(* CODESYS project MariaDB 1.0.1.6.library
   Description: connect to MariaDB read and write simple
      Impressed and helped with OSCAT
      www.oscat.de
   Version: 1.0.1.6
   Title: MariaDB
   Author: Stefan Dreyer
   DocFormat: reStructuredText
   Placeholder: MariaDB
   LanguageModelAttribute: qualified-access-only
   DefaultNamespace: MariaDB
   Company: Stefan Dreyer

Project tree, tasks and I/O mapping:
  libraries: CAA Types Extern, * (CAA Technical Workgroup); CAA Behaviour Model, * (CAA Technical Workgroup); CAA FB Factory, * (CAA Technical Workgroup); Time and Date, 3.5.7.0 (3S - Smart Software Solutions GmbH); SysFile, * (System); SysTypes Interfaces, * (System); Standard, * (System); SysMem, 3.5.12.0 (System); SysSocket, 3.5.15.0 (System); CmpErrors2 Interfaces, 3.5.15.0 (System); Raspberry I2C MUX, 1.0.1.2 (Stefan Dreyer); SysProcess, 3.5.16.0 (System); SysSem, 3.5.16.0 (System); Base Interfaces, 3.5.2.0 (System); BASIC, 3.3.4.0 (OSCAT); OSCAT Network Types, 1.0.0.2 (Stefan Dreyer); Common Helper for development, 1.1.0.6 (Stefan Dreyer); PRO JSON, 1.0.0.12 (Pro Electric)
  MariaDb/
    Structs/
      data type DATA_TO_DB
      data type VALUE_TO_DB_DATA_OFFLINE
      data type DB_SQL_DATA
      data type DATA_FROM_DB
      data type DB_IN_OUT
      data type SQL_ERROR
      data type PARAMETER_DB_DATA
      data type DATA_FOR_VALUE
      data type LOGGING_DATA
      data type COUNTER_TO_DB_DATA
    Function Blocks/
      function block HANDLE_SQL_DB [ST]: SQL_RESPONSE_COMMON
      function block VALUE_TO_DB [ST]: PUSH_LOCAL_BUFFER, SET_DB_REQUEST_FOR_PW_CONFIG, CHECK_DATA_FROM_DB, DO_SQL_DATA, SET_CONFIG_VALUE
      function block TIME_DATE_IMPULS [ST]
      function block MARIADB_CONTROL [ST]
      function block SQL_BASE [ST]: PUT_SQL_TO_BUFFER, CREATE_SQL, SAVE_SQL_ERROR, GET_INDEX_DATA_FIELDS_SQL_RESPONSE, CHECK_EOF_PAKET, DO_SQL_DATA, SET_DB_IN_OUT_PTR
      function block LOGGING_TO_DB [ST]: DO_SQL_DATA, PUSH_LOCAL_BUFFER, SetConfig
      function block PARAMETER_DB [ST]: CHECK_DIFF_VAR, DO_SQL_DATA, GET_PAGE_ADRESS_EEPROM, CHECK_DATA_FROM_DB, CHECK_DATA_FROM_EEPROM
      function block STRING_DB [ST]: CHECK_DIFF_VAR, DO_SQL_DATA, GET_PAGE_ADRESS_EEPROM, CHECK_DATA_FROM_DB, CHECK_DATA_FROM_EEPROM
      function block COUNTER_DB [ST]: SET_CONFIG_COUNTER, PUSH_LOCAL_BUFFER, DO_SQL_DATA
      function block VALUE_TO_DB_AUTO_ID [ST]: PUSH_LOCAL_BUFFER, SET_DB_REQUEST_FOR_PW_CONFIG, CHECK_DATA_FROM_DB, DO_SQL_DATA, SET_CONFIG_VALUE, SET_CONFIG_VALUE_LEVELS, SetRealFaktor
      function block LOGGING_TO_DB_AUTO_ID [ST]: DO_SQL_DATA, PUSH_LOCAL_BUFFER, CHECK_DATA_FROM_DB, SET_DB_REQUEST_FOR_TEXT_CONFIG
      function block VALUE_TO_DB_AUTO_ID_ANY [ST]: PUSH_LOCAL_BUFFER, SET_DB_REQUEST_FOR_PW_CONFIG, CHECK_DATA_FROM_DB, DO_SQL_DATA, SET_CONFIG_VALUE, SET_CONFIG_VALUE_LEVELS
      function block VALUE_TO_DB_AUTO_ID_JSON [ST]: FB_Init
      function block COUNTER_DB_AUTO_ID [ST]: SET_CONFIG_COUNTER, PUSH_LOCAL_BUFFER, DO_SQL_DATA, CHECK_DATA_FROM_DB, SET_DB_REQUEST_FOR_COUNTER_NUM
    GlobalConstants/
      global variables MyConstants
    Types/
      data type SQL_COMMANDS
      data type MYSQL_COM
      data type DB_RESPONSE
    Functions/
      function GET_STRING_DATE [ST]
      function GET_STRING_FROM_RESPONSE [ST]
*)

// MariaDb/Structs/DATA_TO_DB
TYPE DATA_TO_DB :

STRUCT
	//ID of SQL FB to store or of request form DB
	FB_ID:UINT;
	//SQL number
	SQL_NO: INT;//Number of SQL
	//SQL for DB
	SQL_STRING:STRING(MyConstants.COM_STRING_SIZE);
END_STRUCT
END_TYPE

// MariaDb/Structs/VALUE_TO_DB_DATA_OFFLINE
TYPE VALUE_TO_DB_DATA_OFFLINE :
STRUCT
	VALUE:CommonTypesAndFunctions.ALL_TYPES_UNION;
	VALUE_TIME:DT;
END_STRUCT
END_TYPE

// MariaDb/Types/SQL_COMMANDS
{attribute 'qualified_only'}
{attribute 'strict'}
TYPE SQL_COMMANDS :
(
	SEND_PW := 0, SEND_REQUEST_GET_PW_CONFIG := 1, WRITE_LOGGING_TEXT := 2, GET_PARAMETER_VALUE := 3, SET_PARAMETER_VALUE := 4,
	GET_PARAMETER_STRING := 5, SET_PARAMETER_STRING := 6, PUT_COUNTER_TO_DB := 7, PUT_COUNTER_TO_DB_WITH_FACTOR := 8,
	SEND_REQUEST_GET_PW_CONFIG_INSTANCE_NAME := 9, GET_LOGGING_TEXT := 10, CREATE_NEW_SENSOR_ENTRY := 11,
	CREATE_NEW_TEXT_ENTRY := 12, SEND_PW_PROZEDUR := 13, SEND_COUNTER_PROZEDUR := 14, GET_COUNTER_NUM := 15,
	CREATE_NEW_COUNTER_ENTRY := 16
);
END_TYPE

// MariaDb/Structs/DB_SQL_DATA
TYPE DB_SQL_DATA :
STRUCT
//All Infos for an SQL Insert/request for very small SQL!
SQL_TEMPLATE:STRING(255);
SQL_KEYWORDS:ARRAY[0..MyConstants.SQL_MAX_KEYWORDS] OF STRING;
SQL_RESPONSE_FIELDS:INT;//Zero means no Answer expected

END_STRUCT
END_TYPE

// MariaDb/Types/MYSQL_COM
TYPE MYSQL_COM :
STRUCT
	S_BUF : OSCAT_NETWORK_TYPES.NETWORK_BUFFER;
	R_BUF : OSCAT_NETWORK_TYPES.NETWORK_BUFFER;
	SQL_CON : BOOL;
	SQL_URL : STRING(OSCAT_BASIC.STRING_LENGTH);
	SQL_PACKET_NO : BYTE;
	TIMEOUT : TIME;
	DNS_IP4 : DWORD;
	SQL_RCV_STATE : BYTE;
	ERROR_C : DWORD;
	ERROR_T : BYTE;
	RESPONSE : POINTER TO STRING;//pointer for String for Response
	RESPONSE_SIZEOF:UINT;//Max Size of String
	
(* revision history
ks	27. oct. 2012	rev 1.0
	original version
*)
(*
Update from Stefan Dreyer for prozessing responses
01.05.2017
*)
END_STRUCT
END_TYPE

// MariaDb/Structs/DATA_FROM_DB
TYPE DATA_FROM_DB :
STRUCT
	FB_ID:UINT;//ID of SQL Data
	//SQL number
	SQL_NO: INT;
	RESPONSE_TYPE:INT;//Type of response
	DATA_FROM_DB:ARRAY[0..OSCAT_NETWORK_TYPES.NETWORK_BUFFER_LONG_SIZE]OF BYTE;
	SQL_ERROR:SQL_ERROR;
END_STRUCT
END_TYPE

// MariaDb/Structs/DB_IN_OUT
TYPE DB_IN_OUT :
STRUCT
	IN:DATA_TO_DB;
	OUT:DATA_FROM_DB;
	IMP:BOOL;//1s impulse
	SYSTEM_TIME:DT;//Time on SYSTEM
	TIME_IO:BOOL;//TIME IS I.O.
	SQL_CONNECTED:BOOL;
	FB_NO_AUTO:UINT;//
	TD_TIME:OSCAT_BASIC.SDT;
	pendingData:UDINT;
END_STRUCT
END_TYPE

// MariaDb/Types/DB_RESPONSE
{attribute 'qualified_only'}
{attribute 'strict'}
TYPE DB_RESPONSE :
(
	ERROR := -1, OK := 1, DATA_RETURNED := 2
);
END_TYPE

// MariaDb/Structs/SQL_ERROR
TYPE SQL_ERROR :
STRUCT
	SQL_ERROR:STRING(255);//SQL ERROR FROM DB
	SQL_NO:INT;
	SQL_ERROR_TIME:DT;
END_STRUCT
END_TYPE

// MariaDb/Structs/PARAMETER_DB_DATA
TYPE PARAMETER_DB_DATA:
STRUCT
	DATA_EEPROM:CommonTypesAndFunctions.EEPROM_DATA;
	STRING_COUNT:UINT := 200;
	HAS_DB: BOOL;
	HAS_EEPROM: BOOL;
	DB_HAS_PRIORITY: BOOL;
	EEPROM_HAS_PRIORITY: BOOL;

END_STRUCT
END_TYPE

// MariaDb/Structs/DATA_FOR_VALUE
TYPE DATA_FOR_VALUE :
STRUCT
	//name aof Value
	Name:STRING[30];
	//Value itself
	Value: CommonTypesAndFunctions.ALL_TYPES_UNION;
	//type of this value
	TypeOfValue:IBaseLibrary.TypeClass;
	//Number of Value in DB
	ValueNum:UINT;
	//Impulse for value
	ImpValue:BOOL;
END_STRUCT
END_TYPE

// MariaDb/Structs/LOGGING_DATA
TYPE LOGGING_DATA :
STRUCT
	//Time of event
	TimeToLog:DT;
	//positiv or negativ edge
	POrN:BOOL;
	
END_STRUCT
END_TYPE

// MariaDb/Structs/COUNTER_TO_DB_DATA
TYPE COUNTER_TO_DB_DATA :
STRUCT
	VALUE_TIME:DT;
END_STRUCT
END_TYPE

// MariaDb/GlobalConstants/MyConstants
{attribute 'qualified_only'}
VAR_GLOBAL CONSTANT
	FB_BUFFER_SIZE:UINT:=20000;
	COM_STRING_SIZE:UINT:=255;
	SQL_MAX_KEYWORDS:UINT:=10;
	SQL_KEYWORDS_SIZE:UINT:=20;
	SQL_DATA_BUFFER_SIZE:UINT:=200;
	NETWORK_BUFFER_LONG_SIZE:UINT:=4095;
	SQL_RESPONSE_MAX_STRING_SIZE:UINT:=200;
	SQL_LENGTH_FIELD_PAKET:UINT:=5;
	SQL_SIZE_OF_HEADER:UINT:=4;
	SQL_SIZE_OF_EOF_PAKET:UINT:=9;
	SQL_OFFSET_DATA_PAKET:UINT:=4;
SQLS: ARRAY[0..16] OF DB_SQL_DATA:=[
					(*0*)
					(SQL_TEMPLATE:='insert into home.allsensors values("valueWhen", SENSOR, VALUE)',
					SQL_KEYWORDS := ['valueWhen','SENSOR','VALUE'], SQL_RESPONSE_FIELDS := 0),
					(*1*)
					(SQL_TEMPLATE:='select intervall, factor, deltaVar from home.sensors where sensorNum = SENSOR',
					SQL_KEYWORDS := ['SENSOR'], SQL_RESPONSE_FIELDS := 3),
					(*2*)
					(SQL_TEMPLATE:='insert into home.logging(textWhen, text, id_text) values("WHEN1", "TEXT", "ID_TEX_T")',
					SQL_KEYWORDS := ['WHEN1', 'TEXT','ID_TEX_T'], SQL_RESPONSE_FIELDS := 0),
					(*3*)
					(SQL_TEMPLATE:='select value from home.param_value where INDEX = INDEX_NO',
					SQL_KEYWORDS := ['INDEX_NO'], SQL_RESPONSE_FIELDS := 1),
					(*4*)
					(SQL_TEMPLATE:='replace into home.param_value values(INDEX, VALUE)',
					SQL_KEYWORDS := ['INDEX', 'VALUE'], SQL_RESPONSE_FIELDS := 0),
					(*5*)
					(SQL_TEMPLATE:='select string from home.param_string where INDEX = INDEX_NO',
					SQL_KEYWORDS := ['INDEX_NO'], SQL_RESPONSE_FIELDS := 1),
					(*6*)
					(SQL_TEMPLATE:='replace into home.param_string values(INDEX, "STRING")',
					SQL_KEYWORDS := ['INDEX', 'STRING'], SQL_RESPONSE_FIELDS := 0),
					(*7*)
					(SQL_TEMPLATE:='insert into home.allsensors values("valueWhen", SENSOR, 1)',
					SQL_KEYWORDS := ['valueWhen','SENSOR'], SQL_RESPONSE_FIELDS := 0),
					(*8*)
					(SQL_TEMPLATE:='INSERT INTO home.allsensors(valueWhen, sensor, value) VALUES("valueWhen1", NUM, FACTOR / TIMESTAMPDIFF(SECOND,(SELECT * FROM (SELECT MAX(valueWhen) from home.allsensors WHERE sensor = NUM)t),"valueWhen1"))',
					SQL_KEYWORDS := ['valueWhen1','NUM','FACTOR'], SQL_RESPONSE_FIELDS := 0),
					(*9*)
					(SQL_TEMPLATE:='select intervall, factor, deltaVar, sensorNum from home.sensors where Instance = "FBName"',
					SQL_KEYWORDS := ['FBName'], SQL_RESPONSE_FIELDS := 4),
					(*10*)
					(SQL_TEMPLATE:='select texte.text, texte.index from home.texte where Instance = "FBName"',
					SQL_KEYWORDS := ['FBName'], SQL_RESPONSE_FIELDS := 2),
					(*11*)
					(SQL_TEMPLATE:='INSERT INTO home.sensors(description,sensorNum,INSTANCE,Factor) VALUES("NBEZ",(SELECT*FROM home.nextn),"NINSTANCE","NFAKTOR")',
					SQL_KEYWORDS := ['NBEZ', 'NINSTANCE', 'NFAKTOR'], SQL_RESPONSE_FIELDS := 0),
					(*12*)
					(SQL_TEMPLATE:='INSERT INTO home.texte(TEXT, INSTANCE) VALUES("NTEXT", "NINSTANCE")',
					SQL_KEYWORDS := ['NTEXT', 'NINSTANCE'], SQL_RESPONSE_FIELDS := 0),
					(*13*)
					(SQL_TEMPLATE:='CALL home.InsertValue("valueWhen", SENSOR, VALUE)',
					SQL_KEYWORDS := ['valueWhen', 'SENSOR', 'VALUE'], SQL_RESPONSE_FIELDS := 0),
					(*14*)
					(SQL_TEMPLATE:='CALL home.InsertCounter("valueWhen", SENSOR, FAKTOR)',
					SQL_KEYWORDS := ['valueWhen', 'SENSOR', 'FAKTOR'], SQL_RESPONSE_FIELDS := 1),
					(*15*)
					(SQL_TEMPLATE:='select sensorNum from home.sensors where Instance = "FBName"',
					SQL_KEYWORDS := ['FBName'], SQL_RESPONSE_FIELDS := 1),
					(*16*)
					(SQL_TEMPLATE:='INSERT INTO home.sensors(description,sensorNum,INSTANCE,factor) VALUES("NBEZ",(SELECT*FROM home.nextnc),"NINSTANCE","NFAKTOR")',
					SQL_KEYWORDS := ['NBEZ', 'NINSTANCE', 'NFAKTOR'], SQL_RESPONSE_FIELDS := 0)];
END_VAR

// MariaDb/Function Blocks/HANDLE_SQL_DB
FUNCTION_BLOCK HANDLE_SQL_DB  
VAR_IN_OUT
	SQL_INFO : OSCAT_NETWORK_TYPES.MYSQL_INFO;
	DB_IN_OUT:DB_IN_OUT;
END_VAR
VAR_INPUT
	ENABLE : BOOL;
	URL : STRING(OSCAT_BASIC.STRING_LENGTH);
	TIMEOUT : TIME;
END_VAR
VAR_OUTPUT
	ERROR_C : DWORD;
	ERROR_T : BYTE;
END_VAR
VAR
	DT_Maria:TIME_DATE_IMPULS;
	MARIADB_CONTROL: MARIADB_CONTROL;
	step : INT;
	snd_size : INT;
	sql_command : BYTE;
	next_step : INT;
	i1 : INT;
	i2 : INT;
	size_of_string_in_response:UINT;
	len_paket:UDINT;
	id1:UDINT;
	com: MYSQL_COM;
	
	//ID of FB from request
	FB_ID_REQUEST : UINT;
	//Number of actuel SQL
	AKT_SQL_NO : INT;
	
		
	T_SPS_LAST_REQUEST_STARTET:DWORD;
	TIME_LAST_REQUEST:DWORD;
	TIME_LAST_REQUEST_MIN:DWORD:=16#FFFFFFFF;
	TIME_LAST_REQUEST_MAX:DWORD;
	SQLS_PER_SECOND:DWORD;
	TIME_TO_NEW_REQUEST:DWORD;
	SQLS_DONE_IO:DWORD;
	T_SPS_LAST_REQUEST_FINISHED:DWORD;
	CYCLE_TIME:DWORD;
	LAST_CYCLE_TIME:DWORD;
	pendingData:UDINT;
	
END_VAR


DB_IN_OUT.FB_NO_AUTO := 0;//reset FB number
pendingData:= DB_IN_OUT.pendingData;
DB_IN_OUT.pendingData:= 0; 
CYCLE_TIME := OSCAT_BASIC.T_PLC_MS() - LAST_CYCLE_TIME;
LAST_CYCLE_TIME := OSCAT_BASIC.T_PLC_MS();
//get system time and so one
DT_Maria(
	DB_IN_OUT:= DB_IN_OUT);
DB_IN_OUT.IMP := DT_Maria.IMP;
DB_IN_OUT.SYSTEM_TIME := DT_Maria.DT_OUT;
DB_IN_OUT.TIME_IO := DT_Maria.TIME_VAILID;

CASE step OF

00:	IF ENABLE THEN
		COM.SQL_URL := URL;
		COM.TIMEOUT := TIMEOUT;
		step := 10;
		COM.SQL_CON := TRUE;
		
	END_IF;
10:	IF SQL_INFO.SQL_CONNECTED THEN
		step := 40;
	END_IF;
40:	


	IF DB_IN_OUT.IN.FB_ID > 0 AND step = 40 THEN (* Neue Datenreihe(n) vorhanden *)
		(*insert Dato only in step 40!*)

		//start sql command
		sql_command := BYTE#3;
		//store sql in DB Buffer
		OSCAT_BASIC._STRING_TO_BUFFER(str:=DB_IN_OUT.IN.SQL_STRING,pos:=5,pt:=ADR(COM.S_BUF.BUFFER),size:=SIZEOF(COM.S_BUF.BUFFER)); (* String in puffer kopieren *)
		FB_ID_REQUEST := DB_IN_OUT.IN.FB_ID;
		AKT_SQL_NO := DB_IN_OUT.IN.SQL_NO;
		next_step := 40;
		snd_size := 5 + OSCAT_BASIC.LEN(STR:= DB_IN_OUT.IN.SQL_STRING) ;
		T_SPS_LAST_REQUEST_STARTET := OSCAT_BASIC.T_PLC_MS();
		TIME_TO_NEW_REQUEST := OSCAT_BASIC.T_PLC_MS() - T_SPS_LAST_REQUEST_FINISHED;
	END_IF

	IF NOT  ENABLE THEN 	(* LOG-Trigger verarbeiten *)
		COM.SQL_CON := FALSE; (* MySQL Verbindung beenden *)
		step := 0;
	END_IF;

(* ~~~~~~~~~~~~~~~~~~~~~~ *)

199:IF COM.SQL_RCV_STATE = BYTE#1 THEN (* OK *)
		IF MyConstants.SQLS[AKT_SQL_NO].SQL_RESPONSE_FIELDS > 0 THEN//last sql command was request
			//Parse response
			IF COM.R_BUF.BUFFER[4] = MyConstants.SQLS[AKT_SQL_NO].SQL_RESPONSE_FIELDS THEN
				//response have the right number of fields
				//put recive buffer to out bufferNETWORK_BUFFER_LONG_SIZE
				DB_IN_OUT.OUT.DATA_FROM_DB := COM.R_BUF.BUFFER;
				DB_IN_OUT.OUT.SQL_NO:= AKT_SQL_NO;
				DB_IN_OUT.OUT.FB_ID := FB_ID_REQUEST;
				DB_IN_OUT.OUT.RESPONSE_TYPE := DB_RESPONSE.DATA_RETURNED;
			ELSE	
				//wrong response!
				step := 0;//ERROR
			END_IF

		END_IF
		step := next_step;
		SQLS_DONE_IO := SQLS_DONE_IO + 1;
		SQL_RESPONSE_COMMON(DB_IN_OUT:=DB_IN_OUT);
	ELSIF COM.SQL_RCV_STATE = BYTE#2 THEN  (* FEHLER *)
		//step := 0;
		DB_IN_OUT.OUT.SQL_ERROR.SQL_ERROR := SQL_INFO.SQL_ERROR;
		DB_IN_OUT.OUT.SQL_ERROR.SQL_NO := AKT_SQL_NO;
		DB_IN_OUT.OUT.SQL_ERROR.SQL_ERROR_TIME := DB_IN_OUT.SYSTEM_TIME;
		DB_IN_OUT.OUT.FB_ID := FB_ID_REQUEST;
		DB_IN_OUT.OUT.RESPONSE_TYPE := DB_RESPONSE.ERROR;
		COM.SQL_RCV_STATE := BYTE#1;//recive zurücksetzten
		SQL_RESPONSE_COMMON(DB_IN_OUT:=DB_IN_OUT);
	END_IF;

END_CASE;

(* ########################## *)
(* SQL-Kommando ausführen *)
IF sql_command > BYTE#0 THEN

	COM.S_BUF.SIZE := INT_TO_UINT(snd_size);
	snd_size := 0;
	
	i2 := UINT_TO_INT(COM.S_BUF.SIZE) - 1; (* alle " zeichen mit ' ersetzen *)
	FOR i1 := 5 TO i2 DO
		IF COM.S_BUF.BUFFER[i1] = BYTE#34 THEN
			COM.S_BUF.BUFFER[i1] := BYTE#39;
		END_IF;
	END_FOR;

	COM.S_BUF.BUFFER[4] := sql_command;
	COM.SQL_PACKET_NO := BYTE#255;
	sql_command := BYTE#0;
	step := 199;
END_IF;

(* ########################## *)

MARIADB_CONTROL(COM:= COM, INFO:=SQL_INFO);
ERROR_C := COM.ERROR_C;
ERROR_T := COM.ERROR_T;

IF COM.ERROR_T > BYTE#0 THEN  (* FEHLER *)
	step := 0;
END_IF;
//put status to SQLs
DB_IN_OUT.SQL_CONNECTED := SQL_INFO.SQL_CONNECTED;
(* ########################## *)

(* revision history
ks	20. apr. 2012	rev 1.0
	original version

*)

METHOD SQL_RESPONSE_COMMON : BOOL
VAR_IN_OUT
	DB_IN_OUT:DB_IN_OUT;
END_VAR
VAR_INPUT
END_VAR
//Eingänge zurück setzten
DB_IN_OUT.IN.FB_ID := 0;
DB_IN_OUT.IN.SQL_NO := 0;
TIME_LAST_REQUEST := OSCAT_BASIC.T_PLC_MS() - T_SPS_LAST_REQUEST_STARTET;
T_SPS_LAST_REQUEST_FINISHED := OSCAT_BASIC.T_PLC_MS();
TIME_LAST_REQUEST_MIN := MIN(TIME_LAST_REQUEST, TIME_LAST_REQUEST_MIN);
TIME_LAST_REQUEST_MAX := MAX(TIME_LAST_REQUEST, TIME_LAST_REQUEST_MAX);
SQLS_PER_SECOND := REAL_TO_DWORD(1/(DWORD_TO_REAL(TIME_LAST_REQUEST)/1000));
END_METHOD

END_FUNCTION_BLOCK

// MariaDb/Function Blocks/MARIADB_CONTROL
FUNCTION_BLOCK MARIADB_CONTROL
(*
update for MariaDB an not only insert and update(select with !1! result), by Stefan Dreyer
update für MariaDB um nicht nur insert und update sondern auch select(mit max einer antwort!) zu ermöglichen von Stefan Dreyer
*)
VAR_IN_OUT
	COM : MYSQL_COM;
	INFO : OSCAT_NETWORK_TYPES.MYSQL_INFO;
END_VAR
VAR_OUTPUT
END_VAR
VAR
	IP_C : CommonTypesAndFunctions.IP_C_EXT;
	URL_DATA : OSCAT_NETWORK_TYPES.url;
	IPC : CommonTypesAndFunctions.IP_CONTROL;

	step : INT;
	snd_step : INT;
	TON_WAIT : OSCAT_BASIC.TON;
	last_step : INT;
	idx1 : INT;
	idx2 : INT;
	idx3 : INT;
	dw_tmp : DWORD;
	timeout1 : TIME;
	timeout2 : TIME;
	ip_c_red_disable : BOOL;
	auth_password : STRING(64);
	auth_run : BOOL;
	MYSQL_AUTH : OSCAT_NETWORK_TYPES.MYSQL_AUTH;
	scramble1_buffer : ARRAY [0..19] OF BYTE;
	scramble2_buffer : ARRAY [0..19] OF BYTE;
	charset_number : BYTE := 16#08;
	max_packet_size : DWORD := 1024;
	client_flags : DWORD := 16#0003_8601;
	sResultIP : STRING; // IP-Address behind hostname
	(*
	LOG_MSG : LOG_MSG;
	_debug_enable : BOOL := TRUE;
	*)

	nop: INT;
END_VAR

(*
version 1.0		16. apr. 2012
programmer		ks
tested by		ks

MYSQL_CONTROL führt einen SQL Befehl auf einem MySQL-Server durch 
*)

IF com.ERROR_C <> 0 THEN
 step := step;
END_IF 

CASE step OF

00:	IF COM.SQL_CON THEN
		timeout1 := MAX(T#10s,COM.TIMEOUT);
		timeout2 := timeout1 + T#1s;
		INFO.SQL_ERROR := '';
		COM.ERROR_C := DWORD#0;
		COM.ERROR_T := BYTE#0;
		URL_DATA := OSCAT_NETWORK_TYPES.STRING_TO_URL(STR:=COM.SQL_URL,DEFAULT_PROTOCOL:='',DEFAULT_PATH:='/');
		step := 10;
	END_IF;

10:	IF CommonTypesAndFunctions.ResolveIPAddr(sHost:= URL_DATA.DOMAIN, sIPResult:= ADR(sResultIP)) = CmpErrors.Errors.ERR_OK THEN
		step := 20;
	ELSE
		step := 980;
	END_IF

20:	(* MariaDB Steuerkanal einrichten *)
	IF URL_DATA.PORT = WORD#0 THEN
		URL_DATA.PORT := WORD#3306; (* Standard Port *)
	END_IF;
	IP_C.C_PORT := URL_DATA.PORT; (* Portnummer eintragen *)
  	IP_C.C_IP := OSCAT_NETWORK_TYPES.IP4_DECODE(sResultIP); (* IP eintragen *)
  	IP_C.C_MODE := BYTE#0; (* Mode: TCP+ACTIV+PORT *)
  	IP_C.TIME_RESET := TRUE; (* Zeitueberwachung rücksetzen *)
  	IP_C.C_ENABLE := TRUE; (* Verbindungsaufbau freigeben *)
  	IP_C.R_OBSERVE := TRUE; (* Empfangsueberwachung *)
	COM.R_BUF.SIZE := UINT#0;
	COM.SQL_RCV_STATE := BYTE#0;
	step := 30;

30:	IF COM.SQL_RCV_STATE = BYTE#1 THEN
		INFO.SERVER_PROTOCOL_VERSION := COM.R_BUF.BUFFER[4];

		(* ende markierung von string server_version suchen *)
		idx2 := UINT_TO_INT(COM.R_BUF.SIZE) - 1;
		FOR idx1 := 5 TO idx2 DO
			IF COM.R_BUF.BUFFER[idx1] = BYTE#0 THEN EXIT; END_IF;
		END_FOR;
		idx1 := idx1 + 5; (* terminierung und thread-id überspringen *)

		FOR idx2:=0 TO 7 DO	(* Byte 0-7 *)
			scramble1_buffer[idx2] := COM.R_BUF.BUFFER[idx1];
			idx1 := idx1 + 1;
		END_FOR;
		idx1 := idx1 + 1;
		idx2 := idx1 + 1;
		INFO.SERVER_CAPABILITIES := OSCAT_BASIC.WORD_OF_BYTE(COM.R_BUF.BUFFER[idx2], COM.R_BUF.BUFFER[idx1]);
		idx1 := idx1 + 2;
		INFO.SERVER_LANGUAGE := COM.R_BUF.BUFFER[idx1];
		idx1 := idx1 + 1;
		idx2 := idx1 + 1;
		INFO.SERVER_STATUS := OSCAT_BASIC.WORD_OF_BYTE(COM.R_BUF.BUFFER[idx2], COM.R_BUF.BUFFER[idx1]);
		idx1 := idx1 + 15;

		FOR idx2:=8 TO 19 DO	(* Byte 8-19 *)
			scramble1_buffer[idx2] := COM.R_BUF.BUFFER[idx1];
			idx1 := idx1 + 1;
		END_FOR;

		IF INFO.SERVER_PROTOCOL_VERSION < BYTE#10 THEN  (* Error: protocol version zu niedrig *)
			COM.ERROR_T := BYTE#2;
			COM.ERROR_C := DWORD#1;
			step := 980;
		ELSIF URL_DATA.PASSWORD = '' THEN
			step := 50;
		ELSE
			auth_password := URL_DATA.PASSWORD;
			auth_run := TRUE;
			step := 40;
		END_IF;
	END_IF;

40:	MYSQL_AUTH(RUN:= auth_run,PASSWORD:= auth_password ,MESSAGE:= scramble1_buffer,SCRAMBLE:= scramble2_buffer);
	IF NOT auth_run THEN
		step := 50;
	END_IF;

50: (* Client Authentication Packet *)
	(* Byte 0-3 werden später eingetragen *)
	COM.S_BUF.BUFFER[04] := OSCAT_BASIC.BYTE_OF_DWORD(client_flags, BYTE#0); (* client_flags *)
	COM.S_BUF.BUFFER[05] := OSCAT_BASIC.BYTE_OF_DWORD(client_flags, BYTE#1);
	COM.S_BUF.BUFFER[06] := OSCAT_BASIC.BYTE_OF_DWORD(client_flags, BYTE#2);
	COM.S_BUF.BUFFER[07] := OSCAT_BASIC.BYTE_OF_DWORD(client_flags, BYTE#3);
	COM.S_BUF.BUFFER[08] := OSCAT_BASIC.BYTE_OF_DWORD(max_packet_size, BYTE#0); (* max_packet_size *)
	COM.S_BUF.BUFFER[09] := OSCAT_BASIC.BYTE_OF_DWORD(max_packet_size, BYTE#1);
	COM.S_BUF.BUFFER[10] := OSCAT_BASIC.BYTE_OF_DWORD(max_packet_size, BYTE#2);
	COM.S_BUF.BUFFER[11] := OSCAT_BASIC.BYTE_OF_DWORD(max_packet_size, BYTE#3);
	COM.S_BUF.BUFFER[12] := charset_number; (* charset_number *)
	FOR idx1 := 13 TO 35 DO (* 23 bytes filler always 0x00.. *)
		COM.S_BUF.BUFFER[idx1] := BYTE#0;
	END_FOR;
	idx3 := OSCAT_BASIC.LEN(URL_DATA.USER);
	FOR idx2 :=1 TO idx3 DO
		COM.S_BUF.BUFFER[idx1] := OSCAT_BASIC.CODE(URL_DATA.USER, idx2);
		idx1 := idx1 + 1;
	END_FOR;
	COM.S_BUF.BUFFER[idx1] := BYTE#0; (* String terminierung eintragen *)
	idx1 := idx1 + 1;
	IF OSCAT_BASIC.LEN(URL_DATA.PASSWORD) = 0 THEN
		COM.S_BUF.BUFFER[idx1] := BYTE#0; (* scramble_buff length *)
	ELSE
		COM.S_BUF.BUFFER[idx1] := BYTE#20; (* scramble_buff length *)
		FOR idx2 :=0 TO 19 DO
			idx1 := idx1 + 1;
			COM.S_BUF.BUFFER[idx1] := scramble2_buffer[idx2];
		END_FOR;
	END_IF;
	COM.S_BUF.SIZE  := INT_TO_UINT(idx1 + 1); (* Sendelänge eintragen *)

	step := 60;

60:	IF COM.SQL_RCV_STATE = BYTE#1 THEN
		INFO.SQL_CONNECTED := TRUE;
		step := 300;
	END_IF;

(* ================================================== *)

300:	step := UINT_TO_INT(SEL(COM.SQL_CON,700,310)); (* Schritt-Selektion *)

310:	step := 300; (* dummy step *)

(* ================================================== *)

700: (* COM_QUIT *)
	COM.S_BUF.BUFFER[04] := BYTE#1; (* 0x01 COM_QUIT mysql_close *)
	COM.S_BUF.SIZE := UINT#5; (* Sendelänge eintragen *)
	COM.SQL_PACKET_NO := BYTE#255;
	ip_c_red_disable := TRUE;
	step := 710;

710:	IF IP_C.C_STATE = BYTE#0 THEN (* Verbindung durch SQL-Server beendet ? *)
		step := 980;
	END_IF;

(* ================================================== *)

980:IP_C.C_ENABLE := FALSE; (* MYSQL Steuerkanal schliessen *)
	ip_c_red_disable := FALSE;
	INFO.SQL_CONNECTED := FALSE;
	//COM.SQL_CON := FALSE;
	COM.S_BUF.SIZE := UINT#0;
	COM.R_BUF.SIZE := UINT#0;
	snd_step := 0;
	step := 990;
	(*####################  DEBUG-MESSAGE  ###################################*)
	(*IF _debug_enable THEN
		LOG_CL.NEW_MSG := 'QUIT: ERROR CODE >~1< TYPE >~2<';
		LOG_CL.PRINTF[1] := DWORD_TO_STRH(COM.ERROR_C);
		LOG_CL.PRINTF[2] := BYTE_TO_STRING(COM.ERROR_T);
		LOG_MSG();
	END_IF;*)
	(*########################################################################*)

990:IF IP_C.C_STATE = BYTE#0 THEN
		step := 0;
	END_IF;

END_CASE;

(* ++++++++++++++++++++++++++++++++++++++++++++++++++++++++++ *)

IF step >= 30 THEN
	IF COM.R_BUF.SIZE >= UINT#3 AND COM.SQL_RCV_STATE = BYTE#0 THEN (* Daten wurden empfangen ? *)
		(*hier Prüfung für OK und ERROR Paket, immer nur ein Paket*)
		(*Zu erledigen, Error an SQL Ersteller zurück liefern und SQL Verbindung nicht trennen*)
		IF DWORD_TO_UINT(OSCAT_BASIC.DWORD_OF_BYTE(BYTE#0, COM.R_BUF.BUFFER[2], COM.R_BUF.BUFFER[1], COM.R_BUF.BUFFER[0])) + UINT#4 = COM.R_BUF.SIZE THEN
			COM.SQL_PACKET_NO := COM.R_BUF.BUFFER[3];
			IF COM.R_BUF.BUFFER[4] = BYTE#16#FF THEN
				idx2 := 13; (* Error String - Erstes Zeichen *)
				idx3 := UINT_TO_INT(COM.R_BUF.SIZE) - 1; (* Error String - Letztes Zeichen *)
				FOR idx1 := idx2 TO idx3 DO (* alle ' durch ´ ersetzen *)
					IF COM.R_BUF.BUFFER[idx1] = BYTE#39 THEN
						COM.R_BUF.BUFFER[idx1] := BYTE#96;
					END_IF;
				END_FOR;
				INFO.SQL_ERROR := OSCAT_BASIC.BUFFER_TO_STRING(PT:=ADR(COM.R_BUF.BUFFER),SIZE:=COM.R_BUF.SIZE,START:=INT_TO_UINT(idx2),STOP:=INT_TO_UINT(idx3));
				COM.SQL_RCV_STATE := BYTE#2;
				COM.R_BUF.SIZE := UINT#0; (* Empfangsbuffer nach Fehler rücksetzen *)
				
			ELSE
				(*hier OK Paket*)
				COM.SQL_RCV_STATE := BYTE#1;
				(*####################  DEBUG-MESSAGE  ###################################*)
				(*IF _debug_enable THEN
					LOG_CL.NEW_MSG := 'RCV: size >~1<';
					LOG_CL.PRINTF[1] := UINT_TO_STRING(COM.R_BUF.SIZE);
					LOG_MSG();
				END_IF;*)
				(*########################################################################*)
			END_IF;
		ELSE
		//hier mehr Paket Antworten bearbeite.	
		//Parsen der Antworten je nach request

		//Hier oder im Aufruf????  
		//Abarbeitung im Aufruf

		END_IF;
		IF DWORD_TO_UINT(OSCAT_BASIC.DWORD_OF_BYTE(BYTE#0, COM.R_BUF.BUFFER[2], COM.R_BUF.BUFFER[1], COM.R_BUF.BUFFER[0])) = 1 THEN//recived response with data
			COM.SQL_RCV_STATE := BYTE#1;
			
		
		END_IF;
		IP_C.R_OBSERVE := FALSE;
	END_IF;
END_IF;

(* automatisches Datensenden *)

CASE snd_step OF

00:	IF step >= 20 AND COM.S_BUF.SIZE > UINT#0 THEN
		dw_tmp := UINT_TO_DWORD(COM.S_BUF.SIZE - UINT#4); (* packet_length *)
		COM.S_BUF.BUFFER[0] := OSCAT_BASIC.BYTE_OF_DWORD(dw_tmp, BYTE#0);
		COM.S_BUF.BUFFER[1] := OSCAT_BASIC.BYTE_OF_DWORD(dw_tmp, BYTE#1);
		COM.S_BUF.BUFFER[2] := 0;
		COM.SQL_PACKET_NO := COM.SQL_PACKET_NO + 1;
		COM.S_BUF.BUFFER[3] := COM.SQL_PACKET_NO;

		IP_C.R_OBSERVE := TRUE;
		COM.R_BUF.SIZE := UINT#0; (* Empfangsbuffer rücksetzen *)
		COM.SQL_RCV_STATE := BYTE#0;

	        (*####################  DEBUG-MESSAGE  ###################################*)
	        (*IF _debug_enable THEN
	          LOG_CL.NEW_MSG := 'SND: size >~1<';
	          LOG_CL.PRINTF[1] := UINT_TO_STRING(COM.S_BUF.SIZE);
	          LOG_MSG();
	        END_IF;*)
	        (*########################################################################*)

		snd_step := 10;
	END_IF;

10:	IF COM.S_BUF.SIZE = UINT#0 THEN (* warten bis alle daten gesendet sind *)
		snd_step := 0;
	END_IF;

END_CASE;

(* Globale Fehlerbehandlung für Haupt-Routine *)
IF COM.ERROR_T = BYTE#0 AND step > 20 THEN (* noch kein Fehler gespeichert und Hauptroutine aktiv *)
	IF IP_C.ERROR > DWORD#0 AND IP_C.C_ENABLE AND NOT IP_C.TIME_RESET THEN  (* IP Control *)
		IF ip_c_red_disable = FALSE OR IP_C.ERROR <> DWORD#16#FD000000 THEN
			COM.ERROR_C := IP_C.ERROR;
			COM.ERROR_T := BYTE#2;
			step := 980;
		END_IF;
	END_IF;
END_IF;

IF TON_WAIT.Q THEN (* Ablaufstörung - Schrittkette *)
	COM.ERROR_C := INT_TO_DWORD(step); (* aktuellen Schritt eintragen *)
	COM.ERROR_T := BYTE#5;
	step := 980;
END_IF;

(* ######################################################## *)

IPC(IP:= DWORD#0, PORT:= WORD#0 , TIME_OUT:= timeout1, IP_C:= IP_C, S_BUF:= COM.S_BUF, R_BUF:= COM.R_BUF); (* MYSQL Steuerkanal *)

TON_WAIT(IN:=step = last_step AND step > 0,PT:=timeout2);
last_step := step;


(* revision history
ks	20. apr. 2012	rev 1.0
	original version

*)

END_FUNCTION_BLOCK

// MariaDb/Function Blocks/TIME_DATE_IMPULS
FUNCTION_BLOCK TIME_DATE_IMPULS
VAR_IN_OUT
	DB_IN_OUT:DB_IN_OUT;
END_VAR
VAR_INPUT
END_VAR
VAR_OUTPUT
	DT_OUT:DT; //Date an Time
	IMP: BOOL; //1s impulse
	TIME_VAILID: BOOL := FALSE; //Time is Valid
	TD:OSCAT_BASIC.SDT;
END_VAR
VAR
	RT_SYS:RTCLK.GetDateAndTime;
	RT:OSCAT_BASIC.RTC_2;
	DT_OLD:DT;
	GET_TIME: BOOL := TRUE;
	TIME_READED: BOOL;
	TIMEZONE:RTCLK.PERIODE;
	ReReadTime: BOOL;
	ReReadErrorTime:TON;
	ReReadTimeCycle:TON;
END_VAR

RT_SYS(xExecute := GET_TIME);
IF RT_SYS.xDone THEN
	GET_TIME := FALSE;
	IF	RT_SYS.dtDateAndTime < DT#1980-01-01-00:00:00 THEN
		//Keine Valide Uhr auf Raspi!
		ReReadTime := TRUE;
		TIME_VAILID := FALSE;
	ELSE
		TIME_READED := TRUE;
		TIMEZONE := RT_SYS.eTimezone;
		ReReadTime := FALSE;
		TIME_VAILID := TRUE;
	END_IF
END_IF
//Zykliches neulsesen der Uhrzeit
ReReadTimeCycle(in := (TIME_VAILID AND NOT GET_TIME), PT:= T#30M);
IF ReReadTimeCycle.Q THEN
	GET_TIME := TRUE;//try again to read Time	
END_IF


//Neulesezeit nach Error bearbeiten:
ReReadErrorTime(in:=ReReadTime, pt:=T#1S);
IF ReReadErrorTime.Q THEN
	ReReadTime := FALSE;
	GET_TIME := TRUE;//try again to read Time
END_IF
//Realtime Clock bearbeiten // Setzten
RT(set := TIME_READED, SDT := RT_SYS.dtDateAndTime, OFS := 60, DEN:=TRUE);
TIME_READED := FALSE;
//Date and time from oscat fb
DT_OUT:=RT.LOCAL_DT;
//check for second impuls
IF DT_OLD <> DT_OUT THEN
	DT_OLD := DT_OUT;
	imp := TRUE;
ELSE
	imp := FALSE;
END_IF
//make Time for OSCAT functions
TD := OSCAT_BASIC.DT_TO_SDT(DTI:= DT_OUT);

DB_IN_OUT.IMP := IMP;
DB_IN_OUT.SYSTEM_TIME := DT_OUT;
DB_IN_OUT.TD_TIME := TD;
DB_IN_OUT.TIME_IO := TIME_VAILID;

END_FUNCTION_BLOCK

// MariaDb/Function Blocks/VALUE_TO_DB
(*HOWTO
this function controls the sending of process data to DB.
if the queue to db is full it stors the value and date local.
if this local buffer is full, the request is dropt.
the id of the call aof this function must be greater then 0 for detection if the queue to db is empty

*)


FUNCTION_BLOCK VALUE_TO_DB EXTENDS SQL_BASE
VAR_INPUT
	
END_VAR
VAR_OUTPUT
END_VAR
VAR_IN_OUT
	
END_VAR
VAR
	//pointer to extern value
	PointerToValue:CommonTypesAndFunctions.ALL_TYPES_UNION_POINTER;
	
	//Value itself
	Value:CommonTypesAndFunctions.ALL_TYPES_UNION;
	//Impulse for value
	ImpValue:BOOL;
	//Value Name
	Name:STRING(50);
	//type of this value
	TypeOfValue:IBaseLibrary.TypeClass;
	//Number of Value in DB
	ValueNum:UINT;
	//stored Data from request
	DATA_REQUEST:DATA_TO_DB;
	//buffer for DB Offline
	BUFFER:ARRAY[0..MyConstants.FB_BUFFER_SIZE] OF VALUE_TO_DB_DATA_OFFLINE;
	

	//Delta time
	DELTA_T:UINT := 60;
	//Time var for DELTA_T
	DELTA_T_VAR:UINT;
	//type of var to save
	VAR_TYPE:UINT;
	//delta value
	DeltaVar:UINT:=1;
	//Last value of VAR send to DB
	LAST_VALUE:CommonTypesAndFunctions.ALL_TYPES_UNION;
	//request by time and Value given
	REQUEST_INSERT: BOOL;
	//Faktor for real for fix komma
	RealFaktor:UINT:=1;
	//check config from DB every....s
	CHECK_DB_CONFIG:UINT:=300;
	//var for waiting to check
	CHECK_DB_CONFIG_VAR:UINT;
	
	FL_IMP_TO_DB:R_TRIG;
	// set to true, if config is reaced
	configDone: BOOL;

END_VAR

//set right config status to parent
SQLInvalid := NOT configDone;
SQL_NO:=SQL_COMMANDS.SEND_PW_PROZEDUR;//set SQL no for super^()
SUPER^();
//if not config, then leave, do this after super so we calc correct FB numbers
IF ValueNum = 0 OR NOT DbPointerIo THEN RETURN; END_IF;


//just work when Time is i.o.
IF NOT DB_IN_OUT^.TIME_IO THEN RETURN; END_IF
//get value from pointer
Value := CommonTypesAndFunctions.GetValueFromPointer(PointerToValue:= PointerToValue, TypeOfValue:= TypeOfValue);
//Check if a config request is todo
IF DATA_REQUEST.FB_ID <> 0 AND DB_IN_OUT^.IN.FB_ID = 0 THEN
	DB_IN_OUT^.IN := DATA_REQUEST;
	
	DATA_REQUEST.FB_ID := 0;//delete request
END_IF

CHECK_DATA_FROM_DB();

//no second imp, nothing to do...
IF NOT DB_IN_OUT^.IMP  THEN
	RETURN;
END_IF
SET_DB_REQUEST_FOR_PW_CONFIG();
//check time over or impulse
FL_IMP_TO_DB(CLK:= ImpValue);
IF DELTA_T_VAR >0 THEN
	DELTA_T_VAR := DELTA_T_VAR -1;
	IF NOT FL_IMP_TO_DB.Q THEN
		RETURN;
	END_IF
END_IF
//check delta V
REQUEST_INSERT := CommonTypesAndFunctions.CheckDeltaValue(Value:= Value, DeltaVar:= DeltaVar, Faktor:= RealFaktor, LastValue:= LAST_VALUE, TypeOfValue:= TypeOfValue);
//nothing todo...
IF NOT REQUEST_INSERT THEN RETURN; END_IF
//we have an request, so first set new intervall
DELTA_T_VAR := DELTA_T - 1;

//push every Data to local buffer, may we lose an cycle but we have only on place to db 
//check buffer to DB free
	//push to lokal buffer
	//if buffer is full drop request
IF BUFFER_INDEX < MyConstants.FB_BUFFER_SIZE THEN
	PUSH_LOCAL_BUFFER();
END_IF

REQUEST_INSERT := FALSE;

METHOD PRIVATE PUSH_LOCAL_BUFFER
VAR_INPUT
END_VAR
VAR_IN_OUT
END_VAR
IF BUFFER_INDEX < MyConstants.FB_BUFFER_SIZE - 1 THEN 
	BUFFER[BUFFER_INDEX].value := Value;
	BUFFER[BUFFER_INDEX].value_time := DB_IN_OUT^.SYSTEM_TIME;
	BUFFER_INDEX := BUFFER_INDEX + 1; 
END_IF
IF BUFFER_INDEX > MaxBuffer THEN
	MaxBuffer := BUFFER_INDEX;
END_IF
END_METHOD

METHOD PRIVATE SET_DB_REQUEST_FOR_PW_CONFIG
VAR_IN_OUT
END_VAR
//check if time is over
IF CHECK_DB_CONFIG_VAR > 0 THEN
	CHECK_DB_CONFIG_VAR := CHECK_DB_CONFIG_VAR - 1;
	RETURN;	
END_IF
IF NOT DB_IN_OUT^.SQL_CONNECTED THEN RETURN; END_IF
//set new intervall
CHECK_DB_CONFIG_VAR := CHECK_DB_CONFIG;

//now put the request to DB

SQL_VALUES[0] := UINT_TO_STRING(ValueNum);

DATA_REQUEST := PUT_SQL_TO_BUFFER(SQL_NO:=SQL_COMMANDS.SEND_REQUEST_GET_PW_CONFIG);
END_METHOD

METHOD PRIVATE CHECK_DATA_FROM_DB
VAR_IN_OUT
END_VAR
VAR
	i:UINT;
END_VAR
IF DB_IN_OUT^.OUT.FB_ID = DB_IN_OUT^.FB_NO_AUTO THEN
	//got my request back	
	i := GET_INDEX_DATA_FIELDS_SQL_RESPONSE(src:=ADR(DB_IN_OUT^.OUT.DATA_FROM_DB),SQL_COMMANDS.SEND_REQUEST_GET_PW_CONFIG);
	IF i = 0 THEN 
	
		SQL_ERROR.SQL_ERROR := 'no data to Sensor';

		//SQL I.O. but no data 
	ELSE
		//parse first data
		DELTA_T := LIMIT(1, STRING_TO_WORD(GET_STRING_FROM_RESPONSE(SRC:=ADR(DB_IN_OUT^.OUT.DATA_FROM_DB), SIZE:=SIZEOF(DB_IN_OUT^.OUT.DATA_FROM_DB),I:=i)), 65000);
		//Set var to new value to prevent high times in some cases
		DELTA_T_VAR := LIMIT(1, DELTA_T, DELTA_T_VAR);
		//get faktor for Real values
		RealFaktor := LIMIT(1, STRING_TO_WORD(GET_STRING_FROM_RESPONSE(SRC:=ADR(DB_IN_OUT^.OUT.DATA_FROM_DB), SIZE:=SIZEOF(DB_IN_OUT^.OUT.DATA_FROM_DB),I:=i)),100);
		//get min delta for values
		DeltaVar := LIMIT(1, STRING_TO_WORD(GET_STRING_FROM_RESPONSE(SRC:=ADR(DB_IN_OUT^.OUT.DATA_FROM_DB), SIZE:=SIZEOF(DB_IN_OUT^.OUT.DATA_FROM_DB),I:=i)),1000);
	END_IF
	DB_IN_OUT^.OUT.FB_ID := 0;//delete response
	configDone := TRUE;
END_IF
END_METHOD

METHOD PRIVATE DO_SQL_DATA
VAR_INPUT
END_VAR
SQL_VALUES[0] := GET_STRING_DATE(BUFFER[BUFFER_INDEX].value_time);
SQL_VALUES[1] := UINT_TO_STRING(ValueNum);
SQL_VALUES[2] := CommonTypesAndFunctions.GetValueStringFaktor(VALUE:= BUFFER[BUFFER_INDEX].value, TypeOfValue:= TypeOfValue, RealFaktor:= TO_INT(RealFaktor), DecimalPlace:= 0);
END_METHOD

METHOD SET_CONFIG_VALUE
VAR_INPUT
	//Name of Value
	Name:STRING[50];
	//type of this value
	TypeOfValue:IBaseLibrary.TypeClass;
	//Number of Value in DB
	ValueNum:UINT;
	//pointer to value
	PointerToValue:CommonTypesAndFunctions.ALL_TYPES_UNION_POINTER;
	//Pointer to DB Data
	DB_IN_OUT:POINTER TO DB_IN_OUT;
	
END_VAR
THIS^.Name := Name;
	
THIS^.TypeOfValue:=TypeOfValue;
	
THIS^.ValueNum := ValueNum;

THIS^.PointerToValue := PointerToValue;

THIS^.SET_DB_IN_OUT_PTR(DB_IN_OUT);
END_METHOD

END_FUNCTION_BLOCK

// MariaDb/Function Blocks/SQL_BASE
FUNCTION_BLOCK SQL_BASE
VAR_IN_OUT
	
END_VAR
VAR_OUTPUT
END_VAR
VAR
	//referenz to DB Struct
	DB_IN_OUT:POINTER TO DB_IN_OUT;
	//SQL VALUES for SQL string
	SQL_VALUES:ARRAY[0..MyConstants.SQL_MAX_KEYWORDS-1] OF STRING;
	SQL_ERROR:SQL_ERROR;
	
	//index for use of buffer, point to first empty element
	BUFFER_INDEX:UINT;
	//Number of SQL to do From Child, to do the correct SQL replacment 
	SQL_NO:INT;
	//set to true, if something is missing for SQL replacment, so, you can wait till its done
	SQLInvalid: BOOL:=FALSE;
	//Set to true if get DB Pointer 
	DbPointerIo:BOOL;
	//max use of locak buffer
	MaxBuffer:UINT;
	//Instance name
	MyName:CommonTypesAndFunctions.GetInstanceName;
	//get config name String
	getConfigName:STRING;
	
END_VAR

IF not DbPointerIo THEN RETURN; END_IF
	

DB_IN_OUT^.FB_NO_AUTO := DB_IN_OUT^.FB_NO_AUTO + 1;
//add pending Data
DB_IN_OUT^.pendingData:= DB_IN_OUT^.pendingData + BUFFER_INDEX;
SAVE_SQL_ERROR();//check if i did get an SQL ERROR
IF SQLInvalid THEN RETURN; END_IF
//POP from buffer for all childs
IF BUFFER_INDEX > 0 AND DB_IN_OUT^.IN.FB_ID = 0 THEN
	//here pop buffer
	BUFFER_INDEX := BUFFER_INDEX - 1;
	//call child
	DO_SQL_DATA();
	//call child
	DB_IN_OUT^.IN:=PUT_SQL_TO_BUFFER(SQL_NO:=SQL_NO);
END_IF

METHOD PUT_SQL_TO_BUFFER : DATA_TO_DB
VAR_IN_OUT
END_VAR
VAR_INPUT
	SQL_NO:INT;
END_VAR
PUT_SQL_TO_BUFFER.FB_ID := DB_IN_OUT^.FB_NO_AUTO;
PUT_SQL_TO_BUFFER.SQL_NO := SQL_NO;
PUT_SQL_TO_BUFFER.SQL_STRING := CREATE_SQL(SQL_NO:=SQL_NO);
END_METHOD

METHOD CREATE_SQL : String(255)
VAR_INPUT
	SQL_NO:INT;
END_VAR
VAR
	i:INT;
END_VAR
i := 0;
CREATE_SQL := MyConstants.SQLS[SQL_NO].SQL_TEMPLATE;

WHILE MyConstants.SQLS[SQL_NO].SQL_KEYWORDS[i] <> '' DO
	CREATE_SQL := OSCAT_BASIC.REPLACE_ALL(str:=CREATE_SQL, src:=MyConstants.SQLS[SQL_NO].SQL_KEYWORDS[i], rep:=SQL_VALUES[i]);
	i := i + 1;
END_WHILE
END_METHOD

METHOD SAVE_SQL_ERROR : String(255)
VAR_INPUT
END_VAR
VAR_IN_OUT
END_VAR
IF DB_IN_OUT^.FB_NO_AUTO = DB_IN_OUT^.OUT.FB_ID AND DB_IN_OUT^.OUT.RESPONSE_TYPE = DB_RESPONSE.ERROR THEN
	SQL_ERROR := DB_IN_OUT^.OUT.SQL_ERROR;
	DB_IN_OUT^.OUT.FB_ID := 0;//delete response
END_IF
END_METHOD

METHOD GET_INDEX_DATA_FIELDS_SQL_RESPONSE : uint;//found index, if 0 sql i.o. but no data

VAR_INPUT
	src : POINTER TO ARRAY[0..32767]OF BYTE; 
	ID_REQUEST: INT;
END_VAR

VAR
	id1: UINT;
	i1: INT;
	len_paket: UINT;
END_VAR
//now get index of Values paket
GET_INDEX_DATA_FIELDS_SQL_RESPONSE := 0; //if zero, nothing found
//first search first EOF Paket
id1 := MyConstants.SQL_LENGTH_FIELD_PAKET;//second paket index after number of fields
FOR i1 := 0 TO MyConstants.SQLS[ID_REQUEST].SQL_RESPONSE_FIELDS - 1 DO
	len_paket := DWORD_TO_UINT(OSCAT_BASIC.DWORD_OF_BYTE(BYTE#0, src^[+id1+2], src^[id1+1], src^[id1]));
	id1 := id1 + len_paket + MyConstants.SQL_SIZE_OF_HEADER(*SIZE OF HEADER*);
END_FOR
//now i got through all colum definition pakets
//now im must see an eof paket
//paket size should be 5 and EOF MARKER should be 16#fe
IF CHECK_EOF_PAKET(src:=src, i:=id1) THEN
	id1 := id1 + MyConstants.SQL_SIZE_OF_EOF_PAKET;//Index to next paket, Data Paket
END_IF
//if the next paket is an eof paket, no data have been received
IF NOT CHECK_EOF_PAKET(src:=src, i:=id1) THEN
	GET_INDEX_DATA_FIELDS_SQL_RESPONSE := id1 + MyConstants.SQL_OFFSET_DATA_PAKET;				
END_IF
END_METHOD

METHOD CHECK_EOF_PAKET : bool
VAR_INPUT
	src:POINTER TO ARRAY[0..32000]OF BYTE;
	i:UINT;
END_VAR
CHECK_EOF_PAKET :=src^[i] = BYTE#5  AND src^[i+4] =16#FE;
END_METHOD

METHOD DO_SQL_DATA
VAR_INPUT
END_VAR
//just leave Empty, Overwrite in your implementation
END_METHOD

METHOD SET_DB_IN_OUT_PTR : INT
VAR_INPUT
	DB_IN_OUT:POINTER TO DB_IN_OUT;
END_VAR
THIS^.DB_IN_OUT := DB_IN_OUT;
DbPointerIo := TRUE;
END_METHOD

END_FUNCTION_BLOCK

// MariaDb/Functions/GET_STRING_FROM_RESPONSE
FUNCTION GET_STRING_FROM_RESPONSE : STRING(MyConstants.SQL_RESPONSE_MAX_STRING_SIZE)
VAR_INPUT
	SRC:POINTER TO ARRAY[0..32767]OF BYTE;
	SIZE: UINT;
END_VAR
VAR_IN_OUT
	I:UINT;
END_VAR
VAR
END_VAR

GET_STRING_FROM_RESPONSE := OSCAT_BASIC.BUFFER_TO_STRING(PT:=SRC, SIZE:=SIZE,START:=i+1,STOP:=i+1+(SRC^[i] - 1));
i := i + 1 + SRC^[i];

END_FUNCTION

// MariaDb/Functions/GET_STRING_DATE
FUNCTION GET_STRING_DATE : string
VAR_INPUT
DATE_IN:DT;
END_VAR
VAR
END_VAR

GET_STRING_DATE := DT_TO_STRING(DATE_IN);
GET_STRING_DATE := OSCAT_BASIC.RIGHT(STR := GET_STRING_DATE, SIZE := 19);
GET_STRING_DATE := OSCAT_BASIC.REPLACE(STR1:= GET_STRING_DATE, STR2:= ' ', L:= 1, P:= 11);

END_FUNCTION

// MariaDb/Function Blocks/LOGGING_TO_DB
FUNCTION_BLOCK LOGGING_TO_DB EXTENDS SQL_BASE
VAR_INPUT
	//TRIGGER: BOOL;
	Trigger:BOOL;
END_VAR
VAR_OUTPUT
END_VAR
VAR
	BUFFER:ARRAY[0..MyConstants.FB_BUFFER_SIZE] OF LOGGING_DATA;
	
	P_TRIGGER:Standard.R_TRIG;
	N_TRIGGER:Standard.F_TRIG;
	TextOn :STRING(200);
	TextOff :STRING(200);
	IdTextOn:UINT;
	IdTextOff:UINT;
	

END_VAR

SQL_NO:=SQL_COMMANDS.WRITE_LOGGING_TEXT;//set SQL no for super^()

SUPER^();
//my work isnt vailid without time... or DB Pointer
IF NOT DbPointerIo THEN RETURN; END_IF
IF NOT DB_IN_OUT^.TIME_IO THEN RETURN; END_IF

P_TRIGGER(CLK:= Trigger);
N_TRIGGER(CLK:= Trigger);

IF BUFFER_INDEX < MyConstants.FB_BUFFER_SIZE AND ((P_TRIGGER.Q AND IdTextOn > 0)OR (N_TRIGGER.Q AND IdTextOff > 0)) THEN
	PUSH_LOCAL_BUFFER();
END_IF

METHOD DO_SQL_DATA
VAR_INPUT
END_VAR
SQL_VALUES[0] := GET_STRING_DATE(BUFFER[BUFFER_INDEX].TimeToLog);
IF BUFFER[BUFFER_INDEX].POrN THEN //check if event was positiv or negativ
	SQL_VALUES[1] := TextOn;
	SQL_VALUES[2] := UINT_TO_STRING(IdTextOn);
ELSE
	SQL_VALUES[1] := TextOff;	
	SQL_VALUES[2] := UINT_TO_STRING(IdTextOff);
END_IF
END_METHOD

METHOD PUSH_LOCAL_BUFFER
VAR_INPUT
END_VAR
VAR_IN_OUT
	//DB_IN_OUT:DB_IN_OUT;
END_VAR
IF BUFFER_INDEX < MyConstants.FB_BUFFER_SIZE - 1 THEN
	BUFFER[BUFFER_INDEX].TimeToLog := DB_IN_OUT^.SYSTEM_TIME;
	BUFFER[BUFFER_INDEX].POrN := Trigger;
END_IF

BUFFER_INDEX := BUFFER_INDEX + 1; 

IF BUFFER_INDEX > MaxBuffer THEN
	MaxBuffer := BUFFER_INDEX;
END_IF
END_METHOD

METHOD SetConfig
VAR_INPUT
	TextOn:STRING(200);
	TextOff:STRING(200);

	IdTextOn:UINT;
	IdTextOff:UINT;
END_VAR
THIS^.TextOn := TextOn;
THIS^.TextOff := TextOff;
THIS^.IdTextOn := IdTextOn;
THIS^.IdTextOff := IdTextOff;
END_METHOD

END_FUNCTION_BLOCK

// MariaDb/Function Blocks/PARAMETER_DB
//this FB saves an Parameter to DB and/or to EEPROM

FUNCTION_BLOCK PARAMETER_DB EXTENDS SQL_BASE
VAR_IN_OUT
	PARAM:CommonTypesAndFunctions.ALL_TYPES_UNION;
	PARAM_DATA:PARAMETER_DB_DATA;
END_VAR
VAR_INPUT

	PARAMETER_NO:UINT;

END_VAR
VAR_OUTPUT
	VAR_VAILID:BOOL; //Datwas read by DB or EEPROM
END_VAR
VAR
	LAST_VALUE:CommonTypesAndFunctions.ALL_TYPES_UNION;
	SQL_COMMAND:INT;
	INIT_DONE:BOOL;
	BUFFER:ARRAY[0..0] OF CommonTypesAndFunctions.ALL_TYPES_UNION;
	SAVE_PARAM: BOOL;
	EEPROM_SAVE_DONE: BOOL;
	DB_SAVE_DONE: BOOL;
	LOCAL_PARAM:CommonTypesAndFunctions.ALL_TYPES_UNION;
	
	LOAD_AT_BOOT_DONE: BOOL := FALSE;
	
	VALUE_FROM_DB:CommonTypesAndFunctions.ALL_TYPES_UNION;
	VALUE_FROM_EEPROM:CommonTypesAndFunctions.ALL_TYPES_UNION;
	
	VALUE_FROM_DB_LOADED: BOOL;
	VALUE_FROM_EEPROM_LOADED: BOOL;

	
	LOAD_VALUE_FROM_DB: BOOL;
	LOAD_VALUE_FROM_EEPROM: BOOL;

	pResult:SysSem.RTS_IEC_RESULT;
	
	EEPROM_DATA_REQUESTET: BOOL;

	
	PRIORITY_CHECK_DONE: BOOL;
END_VAR

PARAMETER_NO := PARAMETER_NO + 1;

IF PARAM_DATA.HAS_DB THEN
	
	SQL_NO:=SQL_COMMAND;//set SQL no for super^()
	SUPER^();
END_IF



//save done?
IF (EEPROM_SAVE_DONE OR NOT PARAM_DATA.HAS_EEPROM) AND (DB_SAVE_DONE OR NOT PARAM_DATA.HAS_DB) AND SAVE_PARAM THEN
	SAVE_PARAM := FALSE;
END_IF

//Check if param changed
IF CHECK_DIFF_VAR(PARAM:= PARAM, LAST_VALUE := LAST_VALUE) THEN
	//Parameter changed, set save bit 
	SAVE_PARAM := TRUE;
	//restart save if allready in progress
	DB_SAVE_DONE := FALSE;
	EEPROM_SAVE_DONE := FALSE;
	
END_IF

//do boot stuff
IF NOT LOAD_AT_BOOT_DONE THEN//get VAR VALUES from DB an EEPROM
	PRIORITY_CHECK_DONE := FALSE;
	IF PARAM_DATA.HAS_DB AND NOT LOAD_VALUE_FROM_DB THEN
		LOAD_VALUE_FROM_DB := TRUE;
	END_IF
	IF PARAM_DATA.HAS_EEPROM AND NOT LOAD_VALUE_FROM_EEPROM THEN
		LOAD_VALUE_FROM_EEPROM := TRUE; 
	END_IF
	LOAD_AT_BOOT_DONE := TRUE;
END_IF

//check priority

IF PARAM_DATA.HAS_DB AND PARAM_DATA.HAS_EEPROM AND VALUE_FROM_EEPROM_LOADED AND VALUE_FROM_DB_LOADED AND NOT PRIORITY_CHECK_DONE THEN
	PRIORITY_CHECK_DONE := TRUE;
	IF CHECK_DIFF_VAR(PARAM:= VALUE_FROM_DB, LAST_VALUE := VALUE_FROM_EEPROM) THEN
		SAVE_PARAM := TRUE;
	END_IF
	IF PARAM_DATA.EEPROM_HAS_PRIORITY THEN
		PARAM := VALUE_FROM_EEPROM;
	END_IF
	IF PARAM_DATA.DB_HAS_PRIORITY THEN
		PARAM := VALUE_FROM_DB;
	END_IF
	
	
END_IF

//do db stuff
IF PARAM_DATA.HAS_DB THEN
	//Set save to DB
	IF PARAM_DATA.HAS_DB AND SAVE_PARAM AND NOT DB_SAVE_DONE AND BUFFER_INDEX = 0 THEN
			//do sql stuff
			SQL_COMMAND := SQL_COMMANDS.SET_PARAMETER_VALUE;
			BUFFER_INDEX := 1; //set buffer index fix to 1
			BUFFER[0] := PARAM;
			DB_SAVE_DONE := TRUE;
	END_IF
	//check if DB data is avalible
	CHECK_DATA_FROM_DB(PARAM:=PARAM);
	//Load value from DB
	IF LOAD_VALUE_FROM_DB AND BUFFER_INDEX = 0 AND NOT VALUE_FROM_DB_LOADED THEN
		//do sql stuff
		SQL_COMMAND := SQL_COMMANDS.GET_PARAMETER_VALUE;
		BUFFER_INDEX := 1; //set buffer index fix to 1
	END_IF
END_IF


//do EEPROM stuff?
IF NOT PARAM_DATA.DATA_EEPROM.HANDLE_VALID OR NOT PARAM_DATA.HAS_EEPROM THEN
	//no semaphore? go, leave, run, now!!!
	RETURN;
END_IF

//Save to EEPROM 
IF PARAM_DATA.HAS_EEPROM AND SAVE_PARAM AND NOT EEPROM_SAVE_DONE THEN
	IF SysSem.SysSemEnter(hSem:=PARAM_DATA.DATA_EEPROM.SEMAPHORE) = CmpErrors.Errors.ERR_OK THEN
		IF PARAM_DATA.DATA_EEPROM.FB_NO_IN = 0 THEN
			PARAM_DATA.DATA_EEPROM.FB_NO_IN := PARAMETER_NO;
			PARAM_DATA.DATA_EEPROM.WRITE_VALUE := TRUE;
			PARAM_DATA.DATA_EEPROM.VALUE_IN.LWORD_T := PARAM.LWORD_T;
			PARAM_DATA.DATA_EEPROM.ADDRESS_VALUE := GET_PAGE_ADRESS_EEPROM(DATA:= PARAM_DATA);
			EEPROM_SAVE_DONE := TRUE;
		END_IF	
	END_IF
	SysSem.SysSemLeave(hSem:=PARAM_DATA.DATA_EEPROM.SEMAPHORE);
END_IF
//got something from eeprom?
IF 	EEPROM_DATA_REQUESTET THEN
	IF SysSem.SysSemEnter(hSem:=PARAM_DATA.DATA_EEPROM.SEMAPHORE) = CmpErrors.Errors.ERR_OK THEN
		CHECK_DATA_FROM_EEPROM(DATA_EEPROM:= PARAM_DATA.DATA_EEPROM, PARAM:= PARAM);
		SysSem.SysSemLeave(hSem:=PARAM_DATA.DATA_EEPROM.SEMAPHORE);
	END_IF
END_IF
//save to eeprom
IF LOAD_VALUE_FROM_EEPROM AND NOT PARAM_DATA.DATA_EEPROM.READ_VALUE AND NOT VALUE_FROM_EEPROM_LOADED THEN
	IF SysSem.SysSemEnter(hSem:=PARAM_DATA.DATA_EEPROM.SEMAPHORE) = CmpErrors.Errors.ERR_OK THEN
		IF PARAM_DATA.DATA_EEPROM.FB_NO_IN = 0 THEN
			PARAM_DATA.DATA_EEPROM.READ_VALUE := TRUE;
			PARAM_DATA.DATA_EEPROM.ADDRESS_VALUE := GET_PAGE_ADRESS_EEPROM(DATA:= PARAM_DATA);
			PARAM_DATA.DATA_EEPROM.FB_NO_IN := PARAMETER_NO;
			EEPROM_DATA_REQUESTET := TRUE;
		END_IF 
	END_IF
	SysSem.SysSemLeave(hSem:=PARAM_DATA.DATA_EEPROM.SEMAPHORE);
END_IF

METHOD CHECK_DIFF_VAR : BOOL
VAR_IN_OUT
	PARAM:CommonTypesAndFunctions.ALL_TYPES_UNION;
	LAST_VALUE:CommonTypesAndFunctions.ALL_TYPES_UNION;
END_VAR
VAR_INPUT
	
END_VAR
VAR
	i:UINT;
	p1:POINTER TO BYTE;
	p2:POINTER TO BYTE;
END_VAR

p1 := ADR(PARAM);
p2 := ADR(LAST_VALUE);

FOR i := 0 TO SIZEOF(PARAM) - 1 DO
	IF p1[i] <> p2[i] THEN 
		CHECK_DIFF_VAR := TRUE;
	END_IF
END_FOR


LAST_VALUE := PARAM;
END_METHOD

METHOD DO_SQL_DATA
VAR_INPUT
END_VAR
IF SQL_NO = SQL_COMMANDS.SET_PARAMETER_VALUE THEN
	SQL_VALUES[0] := UINT_TO_STRING(PARAMETER_NO - 1);
	SQL_VALUES[1] := LWORD_TO_STRING(BUFFER[BUFFER_INDEX].LWORD_T);
END_IF

IF SQL_NO = SQL_COMMANDS.GET_PARAMETER_VALUE THEN
	SQL_VALUES[0] := UINT_TO_STRING(PARAMETER_NO - 1);
END_IF
END_METHOD

METHOD GET_PAGE_ADRESS_EEPROM : UINT
VAR_INPUT
	DATA:PARAMETER_DB_DATA;
END_VAR
GET_PAGE_ADRESS_EEPROM := DATA.STRING_COUNT * DATA.DATA_EEPROM.PAGE_SIZE + PARAMETER_NO * sizeof(DATA.DATA_EEPROM.VALUE_IN);
END_METHOD

METHOD CHECK_DATA_FROM_DB
VAR_INPUT
END_VAR
VAR_IN_OUT
	
	PARAM:CommonTypesAndFunctions.ALL_TYPES_UNION;
END_VAR
VAR
	i:UINT;
END_VAR
IF DB_IN_OUT^.OUT.FB_ID = DB_IN_OUT^.FB_NO_AUTO THEN
	//got my request back	
	i := GET_INDEX_DATA_FIELDS_SQL_RESPONSE(src:=ADR(DB_IN_OUT^.OUT.DATA_FROM_DB),SQL_COMMANDS.GET_PARAMETER_VALUE);
	IF i = 0 THEN 
		SQL_ERROR.SQL_ERROR := 'no data to parameter ';
		//SQL I.O. but no data
	LAST_VALUE.LWORD_T := 0;
	VALUE_FROM_DB.LWORD_T := 0;
	 
	ELSE
		//parse first data
		PARAM.LWORD_T := STRING_TO_LWORD(GET_STRING_FROM_RESPONSE(SRC:=ADR(DB_IN_OUT^.OUT.DATA_FROM_DB), SIZE:=SIZEOF(DB_IN_OUT^.OUT.DATA_FROM_DB),I:=i));
		//set laste value to prevent save trigger
		LAST_VALUE := PARAM;
		PARAM := PARAM;
	END_IF
	VALUE_FROM_DB_LOADED := TRUE;
	VAR_VAILID := TRUE;
	DB_IN_OUT^.OUT.FB_ID := 0;//delete response
	LOAD_VALUE_FROM_DB := FALSE;//delete request
END_IF
END_METHOD

METHOD CHECK_DATA_FROM_EEPROM
VAR_IN_OUT
	DATA_EEPROM:CommonTypesAndFunctions.EEPROM_DATA;
	PARAM:CommonTypesAndFunctions.ALL_TYPES_UNION;
END_VAR
IF DATA_EEPROM.FB_NO_OUT = PARAMETER_NO THEN
	//got my request back	

	//get value
	VALUE_FROM_EEPROM.LWORD_T := DATA_EEPROM.VALUE_OUT.LWORD_T;
	IF NOT  VALUE_FROM_DB_LOADED THEN
		PARAM := VALUE_FROM_EEPROM;
		LAST_VALUE := VALUE_FROM_EEPROM;
	
	END_IF 
	
	
	//set laste value to prevent save trigger
	VALUE_FROM_EEPROM_LOADED := TRUE;
	VAR_VAILID := TRUE;
	
	DATA_EEPROM.FB_NO_OUT := 0;//delete response
	LOAD_VALUE_FROM_EEPROM := FALSE;//delete request
	EEPROM_DATA_REQUESTET := FALSE;
END_IF
END_METHOD

END_FUNCTION_BLOCK

// MariaDb/Function Blocks/STRING_DB
//this FB saves an Parameter to DB and/or to EEPROM

FUNCTION_BLOCK STRING_DB EXTENDS SQL_BASE
VAR_IN_OUT
	PARAM:STRING(STRING_SIZE);
	DATA:PARAMETER_DB_DATA;
END_VAR
VAR_INPUT

	PARAMETER_NO:UINT;

END_VAR
VAR_OUTPUT
	VAR_VAILID:BOOL; //Datwas read by DB or EEPROM
END_VAR
VAR
	LAST_VALUE:STRING(STRING_SIZE);
	SQL_COMMAND:INT;
	INIT_DONE:BOOL;
	BUFFER:ARRAY[0..0] OF STRING(STRING_SIZE);
	SAVE_PARAM: BOOL;
	EEPROM_SAVE_DONE: BOOL;
	DB_SAVE_DONE: BOOL;
	LOCAL_PARAM:CommonTypesAndFunctions.ALL_TYPES_UNION;
	
	LOAD_AT_BOOT_DONE: BOOL := FALSE;
	
	VALUE_FROM_DB:STRING(STRING_SIZE);
	VALUE_FROM_EEPROM:STRING(STRING_SIZE);
	
	VALUE_FROM_DB_LOADED: BOOL;
	VALUE_FROM_EEPROM_LOADED: BOOL;

	
	LOAD_VALUE_FROM_DB: BOOL;
	LOAD_VALUE_FROM_EEPROM: BOOL;

	pResult:SysSem.RTS_IEC_RESULT;
	
	EEPROM_DATA_REQUESTET: BOOL;

	
	PRIORITY_CHECK_DONE: BOOL;
END_VAR
VAR CONSTANT
	STRING_SIZE : UINT := 127;
END_VAR

PARAMETER_NO := PARAMETER_NO + 1;
IF DATA.HAS_DB THEN
	
	SQL_NO:=SQL_COMMAND;//set SQL no for super^()
	SUPER^();
END_IF

//save done?
IF (EEPROM_SAVE_DONE OR NOT DATA.HAS_EEPROM) AND (DB_SAVE_DONE OR NOT DATA.HAS_DB) AND SAVE_PARAM THEN
	SAVE_PARAM := FALSE;
END_IF

//Check if param changed
IF CHECK_DIFF_VAR(PARAM:= PARAM, LAST_VALUE := LAST_VALUE) THEN
	//Parameter changed, set save bit 
	SAVE_PARAM := TRUE;
	//restart save if allready in progress
	DB_SAVE_DONE := FALSE;
	EEPROM_SAVE_DONE := FALSE;
	
END_IF
LAST_VALUE := PARAM;
//do boot stuff
IF NOT LOAD_AT_BOOT_DONE THEN//get VAR VALUES from DB an EEPROM
	PRIORITY_CHECK_DONE := FALSE;
	IF DATA.HAS_DB AND NOT LOAD_VALUE_FROM_DB THEN
		LOAD_VALUE_FROM_DB := TRUE;
	END_IF
	IF DATA.HAS_EEPROM AND NOT LOAD_VALUE_FROM_EEPROM THEN
		LOAD_VALUE_FROM_EEPROM := TRUE; 
	END_IF
	LOAD_AT_BOOT_DONE := TRUE;
END_IF

//check priority
IF DATA.HAS_DB AND DATA.HAS_EEPROM AND VALUE_FROM_EEPROM_LOADED AND VALUE_FROM_DB_LOADED AND NOT PRIORITY_CHECK_DONE THEN
	PRIORITY_CHECK_DONE := TRUE;
	//check if params are diffrent
	IF CHECK_DIFF_VAR(PARAM:= VALUE_FROM_EEPROM, LAST_VALUE := VALUE_FROM_DB) THEN
		SAVE_PARAM := TRUE;
	END_IF
	//load priority param
	IF DATA.EEPROM_HAS_PRIORITY THEN
		PARAM := VALUE_FROM_EEPROM;
	END_IF
	IF DATA.DB_HAS_PRIORITY THEN
		PARAM := VALUE_FROM_DB;
	END_IF
END_IF

//do db stuff
IF DATA.HAS_DB THEN
	//Set save to DB
	IF DATA.HAS_DB AND SAVE_PARAM AND NOT DB_SAVE_DONE AND BUFFER_INDEX = 0 THEN
			//do sql stuff
			SQL_COMMAND := SQL_COMMANDS.SET_PARAMETER_STRING;
			BUFFER_INDEX := 1; //set buffer index fix to 1
			BUFFER[0] := PARAM;
			DB_SAVE_DONE := TRUE;
	END_IF
	//check if DB data is avalible
	CHECK_DATA_FROM_DB(PARAM:=PARAM);
	//Load value from DB
	IF LOAD_VALUE_FROM_DB AND BUFFER_INDEX = 0 AND NOT VALUE_FROM_DB_LOADED THEN
		//do sql stuff
		SQL_COMMAND := SQL_COMMANDS.GET_PARAMETER_STRING;
		BUFFER_INDEX := 1; //set buffer index fix to 1
	END_IF
END_IF


//do EEPROM stuff?
IF NOT DATA.DATA_EEPROM.HANDLE_VALID OR NOT DATA.HAS_EEPROM THEN
	//no semaphore? go, leave, run, now!!!
	RETURN;
END_IF

//Save to EEPROM 
IF DATA.HAS_EEPROM AND SAVE_PARAM AND NOT EEPROM_SAVE_DONE THEN
	IF SysSem.SysSemEnter(hSem:=DATA.DATA_EEPROM.SEMAPHORE) = CmpErrors.Errors.ERR_OK THEN
		IF DATA.DATA_EEPROM.FB_NO_IN = 0 THEN
			DATA.DATA_EEPROM.FB_NO_IN := PARAMETER_NO;
			DATA.DATA_EEPROM.WRITE_PAGE := TRUE;
			OSCAT_BASIC._STRING_TO_BUFFER(STR:= PARAM, POS:= 0, PT:= ADR(DATA.DATA_EEPROM.PAGE_IN), SIZE:= INT_TO_UINT( Standard.LEN(STR:= PARAM) + 1));//write the zero to buffer
			DATA.DATA_EEPROM.ADDRESS_PAGE := GET_PAGE_ADRESS_EEPROM(DATA:= DATA);
			EEPROM_SAVE_DONE := TRUE;
		END_IF	
	END_IF
	SysSem.SysSemLeave(hSem:=DATA.DATA_EEPROM.SEMAPHORE);
END_IF
//got something from eeprom?
IF 	EEPROM_DATA_REQUESTET THEN
	IF SysSem.SysSemEnter(hSem:=DATA.DATA_EEPROM.SEMAPHORE) = CmpErrors.Errors.ERR_OK THEN
		CHECK_DATA_FROM_EEPROM(DATA_EEPROM:= DATA.DATA_EEPROM, PARAM:= PARAM);
		SysSem.SysSemLeave(hSem:=DATA.DATA_EEPROM.SEMAPHORE);
	END_IF
END_IF
//save to eeprom
IF LOAD_VALUE_FROM_EEPROM AND NOT DATA.DATA_EEPROM.READ_VALUE AND NOT VALUE_FROM_EEPROM_LOADED THEN
	IF SysSem.SysSemEnter(hSem:=DATA.DATA_EEPROM.SEMAPHORE) = CmpErrors.Errors.ERR_OK THEN
		IF DATA.DATA_EEPROM.FB_NO_IN = 0 THEN
			DATA.DATA_EEPROM.READ_PAGE := TRUE;
			DATA.DATA_EEPROM.ADDRESS_PAGE := GET_PAGE_ADRESS_EEPROM(DATA:= DATA);
			DATA.DATA_EEPROM.FB_NO_IN := PARAMETER_NO;
			EEPROM_DATA_REQUESTET := TRUE;
		END_IF 
	END_IF
	SysSem.SysSemLeave(hSem:=DATA.DATA_EEPROM.SEMAPHORE);
END_IF

METHOD CHECK_DIFF_VAR : BOOL
VAR_IN_OUT
	PARAM:STRING(STRING_SIZE);
	LAST_VALUE:STRING(STRING_SIZE);
END_VAR
IF NOT CommonTypesAndFunctions.StrEquals(ADR(PARAM), ADR(LAST_VALUE)) = 0 THEN
	CHECK_DIFF_VAR := FALSE;
ELSE
	CHECK_DIFF_VAR := TRUE;
END_IF
END_METHOD

METHOD DO_SQL_DATA
VAR_INPUT
END_VAR
//just leave Empty, Overwrite in your implementation

IF SQL_NO = SQL_COMMANDS.SET_PARAMETER_STRING THEN
	SQL_VALUES[0] := UINT_TO_STRING(PARAMETER_NO - 1);
	SQL_VALUES[1] := BUFFER[BUFFER_INDEX];
END_IF

IF SQL_NO = SQL_COMMANDS.GET_PARAMETER_STRING THEN
	SQL_VALUES[0] := UINT_TO_STRING(PARAMETER_NO - 1);
END_IF
END_METHOD

METHOD GET_PAGE_ADRESS_EEPROM : UINT
VAR_INPUT
	DATA:PARAMETER_DB_DATA;
END_VAR
GET_PAGE_ADRESS_EEPROM := DATA.DATA_EEPROM.PAGE_SIZE * (PARAMETER_NO - 1);//
END_METHOD

METHOD CHECK_DATA_FROM_DB
VAR_IN_OUT
	PARAM:STRING(STRING_SIZE);
END_VAR
VAR
	i:UINT;
END_VAR
IF DB_IN_OUT^.OUT.FB_ID = DB_IN_OUT^.FB_NO_AUTO THEN
	//got my request back	
	i := GET_INDEX_DATA_FIELDS_SQL_RESPONSE(src:=ADR(DB_IN_OUT^.OUT.DATA_FROM_DB),SQL_COMMANDS.GET_PARAMETER_VALUE);
	IF i = 0 THEN 
		SQL_ERROR.SQL_ERROR := 'no data to parameter ';
		//SQL I.O. but no data
	LAST_VALUE := '';//start save trigger...
	VALUE_FROM_DB := '';
	 
	ELSE
		//parse first data
		VALUE_FROM_DB := GET_STRING_FROM_RESPONSE(SRC:=ADR(DB_IN_OUT^.OUT.DATA_FROM_DB), SIZE:=SIZEOF(DB_IN_OUT^.OUT.DATA_FROM_DB),I:=i);
		IF NOT VALUE_FROM_EEPROM_LOADED THEN
			//set laste value to prevent save trigger
			LAST_VALUE := VALUE_FROM_DB;
			PARAM := VALUE_FROM_DB;
		END_IF
	END_IF
	VALUE_FROM_DB_LOADED := TRUE;
	VAR_VAILID := TRUE;
	DB_IN_OUT^.OUT.FB_ID := 0;//delete response
	LOAD_VALUE_FROM_DB := FALSE;//delete request
END_IF
END_METHOD

METHOD CHECK_DATA_FROM_EEPROM
VAR_IN_OUT
	DATA_EEPROM:CommonTypesAndFunctions.EEPROM_DATA;
	PARAM:STRING(STRING_SIZE);
END_VAR
VAR 
	i:UINT;
END_VAR
IF DATA_EEPROM.FB_NO_OUT = PARAMETER_NO THEN
	//got my request back	
	
	//search String termination
	FOR  i := 0 TO STRING_SIZE + 1 DO
 		IF DATA_EEPROM.PAGE_OUT[i] = 0 THEN
			EXIT;
		END_IF
	END_FOR	 
	//get value
	
	VALUE_FROM_EEPROM := OSCAT_BASIC.BUFFER_TO_STRING(PT:= ADR(DATA_EEPROM.PAGE_OUT), SIZE:= SIZEOF(DATA_EEPROM.PAGE_OUT), START:=0 , STOP:= i - 1);
	IF NOT VALUE_FROM_EEPROM_LOADED THEN
		PARAM := VALUE_FROM_EEPROM;
		LAST_VALUE := VALUE_FROM_EEPROM;	
	END_IF
	//set laste value to prevent save trigger
	VALUE_FROM_EEPROM_LOADED := TRUE;
	VAR_VAILID := TRUE;
	
	DATA_EEPROM.FB_NO_OUT := 0;//delete response
	LOAD_VALUE_FROM_EEPROM := FALSE;//delete request
	EEPROM_DATA_REQUESTET := FALSE;
END_IF
END_METHOD

END_FUNCTION_BLOCK

// MariaDb/Function Blocks/COUNTER_DB
(*do never ever try to use dynamic divider --> easy count of comsumption is not possible*)
FUNCTION_BLOCK COUNTER_DB EXTENDS SQL_BASE
VAR_INPUT
	//impulse from counter
	imp:BOOL;
END_VAR
VAR_OUTPUT
END_VAR
VAR
	//Counter Name
	Name:STRING(50);
	//Number of counter in DB
	CounterNum:UINT;
	//rising trigger of counter
	TrRis:Standard.R_TRIG;
	//buffer for DB Offline
	BUFFER:ARRAY[0..MyConstants.FB_BUFFER_SIZE] OF COUNTER_TO_DB_DATA;
	//impulses since start
	imps:ULINT;
	//consumption Factor
	LConsumptionFaktor:UDINT;

END_VAR


SUPER^();
//if not config, then leave, do this after super so we calc correct FB numbers
IF CounterNum = 0 OR NOT DbPointerIo THEN RETURN; END_IF;

//just work when Time is i.o.
IF NOT DB_IN_OUT^.TIME_IO THEN RETURN; END_IF

TrRis(CLK:= imp);
//do all work only on rising edge
IF NOT TrRis.Q THEN RETURN; END_IF

imps := imps + 1;

IF BUFFER_INDEX < MyConstants.FB_BUFFER_SIZE THEN
	PUSH_LOCAL_BUFFER();
END_IF

METHOD SET_CONFIG_COUNTER
VAR_INPUT
	//Name of Value
	Name:STRING[50];
	//Number of counter in DB
	CounterNum:UINT;
	//Pointer to DB Data
	DB_IN_OUT:POINTER TO DB_IN_OUT;
	//factor for DB query
	//if 0 don't calculat actualy usage
	consumptionFaktor:UDINT;
END_VAR
THIS^.Name := Name;
		
THIS^.CounterNum := CounterNum;

THIS^.SET_DB_IN_OUT_PTR(DB_IN_OUT);

LConsumptionFaktor := consumptionFaktor;
IF consumptionFaktor= 0 THEN
	SQL_NO:=SQL_COMMANDS.PUT_COUNTER_TO_DB;//set SQL no for super^()
ELSE
	SQL_NO:=SQL_COMMANDS.PUT_COUNTER_TO_DB_WITH_FACTOR;//set SQL no for super^()
END_IF
END_METHOD

METHOD PRIVATE PUSH_LOCAL_BUFFER
VAR_INPUT
END_VAR
VAR_IN_OUT
	//DB_IN_OUT:DB_IN_OUT;
END_VAR
IF BUFFER_INDEX < MyConstants.FB_BUFFER_SIZE - 1 THEN 
	BUFFER[BUFFER_INDEX].value_time := DB_IN_OUT^.SYSTEM_TIME;
	BUFFER_INDEX := BUFFER_INDEX + 1; 
END_IF
IF BUFFER_INDEX > MaxBuffer THEN
	MaxBuffer := BUFFER_INDEX;
END_IF
END_METHOD

METHOD PRIVATE DO_SQL_DATA
VAR_INPUT
END_VAR
VAR
	i:UINT;
	lowest:UINT;
END_VAR
//BUFFER_INDEX points to last valid value, so search the oldest and get this to DB
IF BUFFER_INDEX = 0 THEN
	//if just one item --> don't care
	SQL_VALUES[0] := GET_STRING_DATE(BUFFER[BUFFER_INDEX].value_time);
ELSE
	lowest:= 0;
	FOR i:= 0 TO BUFFER_INDEX DO
		IF BUFFER[i].value_time < BUFFER[lowest].value_time THEN
			lowest:= i; 
		END_IF
	END_FOR
	SQL_VALUES[0] := GET_STRING_DATE(BUFFER[lowest].value_time);
	//now copy last in lowest for consistens
	BUFFER[lowest].value_time:= BUFFER[BUFFER_INDEX].value_time;
END_IF
SQL_VALUES[1] := UINT_TO_STRING(CounterNum);
SQL_VALUES[2] := UDINT_TO_STRING(LConsumptionFaktor);
END_METHOD

END_FUNCTION_BLOCK

// MariaDb/Function Blocks/VALUE_TO_DB_AUTO_ID
(*HOWTO
this function controls the sending of process data to DB.
if the queue to db is full it stors the value and date local.
if this local buffer is full, the request is dropt.
the id of the call aof this function must be greater then 0 for detection if the queue to db is empty
This FB creats datapoints by its names
*)


FUNCTION_BLOCK VALUE_TO_DB_AUTO_ID EXTENDS SQL_BASE
VAR_INPUT

END_VAR
VAR_OUTPUT
END_VAR
VAR_IN_OUT
	
END_VAR
VAR
	//pointer to extern value
	PointerToValue:CommonTypesAndFunctions.ALL_TYPES_UNION_POINTER;
	
	//Value itself
	Value:CommonTypesAndFunctions.ALL_TYPES_UNION;
	//Impulse for value
	ImpValue:BOOL;
	//Value Name
	Name:STRING(50);
	//type of this value
	TypeOfValue:IBaseLibrary.TypeClass;
	//Number of Value in DB
	ValueNum:UINT;
	//stored Data from request
	DATA_REQUEST:DATA_TO_DB;
	//buffer for DB Offline
	BUFFER:ARRAY[0..MyConstants.FB_BUFFER_SIZE] OF VALUE_TO_DB_DATA_OFFLINE;
	

	//Delta time
	DELTA_T:UINT := 60;
	//Time var for DELTA_T
	DELTA_T_VAR:UINT;
	//type of var to save
	VAR_TYPE:UINT;
	//delta value
	DeltaVar:UINT:=1;
	//Last value of VAR send to DB
	LAST_VALUE:CommonTypesAndFunctions.ALL_TYPES_UNION;
	//request by time and Value given
	REQUEST_INSERT: BOOL;
	//Faktor for real for fix komma
	RealFaktor:UINT:=1;
	//check config from DB every....s
	CHECK_DB_CONFIG:UINT:=300;
	//var for waiting to check
	CHECK_DB_CONFIG_VAR:UINT;
	
	FL_IMP_TO_DB:R_TRIG;
	// set to true, if config is reaced
	configDone: BOOL;
	

END_VAR

//set right config status to parent
SQLInvalid := NOT configDone OR valueNum = 0;
SQL_NO:=SQL_COMMANDS.SEND_PW_PROZEDUR;//set SQL no for super^()
SUPER^();
//if not config, then leave, do this after super so we calc correct FB numbers
IF NOT DbPointerIo THEN RETURN; END_IF;


//just work when Time is i.o.
IF NOT DB_IN_OUT^.TIME_IO THEN RETURN; END_IF
//get value from pointer
Value := CommonTypesAndFunctions.GetValueFromPointer(PointerToValue:= PointerToValue, TypeOfValue:= TypeOfValue);
//Check if a config request is todo
IF DATA_REQUEST.FB_ID <> 0 AND DB_IN_OUT^.IN.FB_ID = 0 THEN
	DB_IN_OUT^.IN := DATA_REQUEST;
	
	DATA_REQUEST.FB_ID := 0;//delete request
END_IF

CHECK_DATA_FROM_DB();

//no second imp, nothing to do...
IF NOT DB_IN_OUT^.IMP  THEN
	RETURN;
END_IF
SET_DB_REQUEST_FOR_PW_CONFIG();
//check time over or impulse
FL_IMP_TO_DB(CLK:= ImpValue);
IF DELTA_T_VAR >0 THEN
	DELTA_T_VAR := DELTA_T_VAR -1;
	IF NOT FL_IMP_TO_DB.Q THEN
		RETURN;
	END_IF
END_IF
//check delta V
REQUEST_INSERT := CommonTypesAndFunctions.CheckDeltaValue(Value:= Value, DeltaVar:= DeltaVar, Faktor:= RealFaktor, LastValue:= LAST_VALUE, TypeOfValue:= TypeOfValue);
//nothing todo...
IF NOT REQUEST_INSERT THEN RETURN; END_IF
//we have an request, so first set new intervall
DELTA_T_VAR := DELTA_T - 1;

//push every Data to local buffer, may we lose an cycle but we have only on place to db 
//check buffer to DB free
	//push to lokal buffer
	//if buffer is full drop request
IF BUFFER_INDEX < MyConstants.FB_BUFFER_SIZE THEN
	PUSH_LOCAL_BUFFER();
END_IF

REQUEST_INSERT := FALSE;

METHOD PRIVATE PUSH_LOCAL_BUFFER
VAR_INPUT
END_VAR
VAR_IN_OUT
END_VAR
IF BUFFER_INDEX < MyConstants.FB_BUFFER_SIZE - 1 THEN 
	BUFFER[BUFFER_INDEX].value := Value;
	BUFFER[BUFFER_INDEX].value_time := DB_IN_OUT^.SYSTEM_TIME;
	BUFFER_INDEX := BUFFER_INDEX + 1; 
END_IF
IF BUFFER_INDEX > MaxBuffer THEN
	MaxBuffer := BUFFER_INDEX;
END_IF
END_METHOD

METHOD PRIVATE SET_DB_REQUEST_FOR_PW_CONFIG
VAR_IN_OUT
	
END_VAR
//check if time is over
IF CHECK_DB_CONFIG_VAR > 0 THEN
	CHECK_DB_CONFIG_VAR := CHECK_DB_CONFIG_VAR - 1;
	RETURN;	
END_IF
IF NOT DB_IN_OUT^.SQL_CONNECTED THEN RETURN; END_IF
//set new intervall
CHECK_DB_CONFIG_VAR := CHECK_DB_CONFIG + DB_IN_OUT^.FB_NO_AUTO;
//now put the request to DB
SQL_VALUES[0] := getConfigName;
DATA_REQUEST := PUT_SQL_TO_BUFFER(SQL_NO:=SQL_COMMANDS.SEND_REQUEST_GET_PW_CONFIG_INSTANCE_NAME);
END_METHOD

METHOD PRIVATE CHECK_DATA_FROM_DB
VAR_IN_OUT
END_VAR
VAR
	//DataField Index
	i:UINT;
END_VAR
IF DB_IN_OUT^.OUT.FB_ID = DB_IN_OUT^.FB_NO_AUTO THEN
	//got my request back	
	i := GET_INDEX_DATA_FIELDS_SQL_RESPONSE(src:=ADR(DB_IN_OUT^.OUT.DATA_FROM_DB),SQL_COMMANDS.SEND_REQUEST_GET_PW_CONFIG_INSTANCE_NAME);
	IF i = 0 THEN 
	
		SQL_ERROR.SQL_ERROR := 'no data to Sensor';
		//so create new entry...
		SQL_VALUES[0] := getConfigName;
		SQL_VALUES[1] := getConfigName;
		SQL_VALUES[2] := TO_STRING(RealFaktor);
		DATA_REQUEST := PUT_SQL_TO_BUFFER(SQL_NO:=SQL_COMMANDS.CREATE_NEW_SENSOR_ENTRY);
		//SQL I.O. but no data 
	ELSE
		//parse first data
		DELTA_T := LIMIT(1, STRING_TO_WORD(GET_STRING_FROM_RESPONSE(SRC:=ADR(DB_IN_OUT^.OUT.DATA_FROM_DB), SIZE:=SIZEOF(DB_IN_OUT^.OUT.DATA_FROM_DB),I:=i)), 65000);
		//Set var to new value to prevent high times in some cases
		DELTA_T_VAR := LIMIT(1, DELTA_T, DELTA_T_VAR);
		//get faktor for Real values
		RealFaktor := LIMIT(1, STRING_TO_WORD(GET_STRING_FROM_RESPONSE(SRC:=ADR(DB_IN_OUT^.OUT.DATA_FROM_DB), SIZE:=SIZEOF(DB_IN_OUT^.OUT.DATA_FROM_DB),I:=i)),100);
		//get min delta for values
		DeltaVar := LIMIT(1, STRING_TO_WORD(GET_STRING_FROM_RESPONSE(SRC:=ADR(DB_IN_OUT^.OUT.DATA_FROM_DB), SIZE:=SIZEOF(DB_IN_OUT^.OUT.DATA_FROM_DB),I:=i)),1000);
		//Get sensor Num
		ValueNum := LIMIT(1, STRING_TO_WORD(GET_STRING_FROM_RESPONSE(SRC:=ADR(DB_IN_OUT^.OUT.DATA_FROM_DB), SIZE:=SIZEOF(DB_IN_OUT^.OUT.DATA_FROM_DB),I:=i)), 65000);
		configDone := TRUE;
	END_IF
	DB_IN_OUT^.OUT.FB_ID := 0;//delete response
	
END_IF
END_METHOD

METHOD PRIVATE DO_SQL_DATA
VAR_INPUT
END_VAR
SQL_VALUES[0] := GET_STRING_DATE(BUFFER[BUFFER_INDEX].value_time);
SQL_VALUES[1] := UINT_TO_STRING(ValueNum);
SQL_VALUES[2] := CommonTypesAndFunctions.GetValueStringFaktor(VALUE:= BUFFER[BUFFER_INDEX].value, TypeOfValue:= TypeOfValue, RealFaktor:= TO_INT(RealFaktor), DecimalPlace:= 0);
END_METHOD

METHOD SET_CONFIG_VALUE
VAR_INPUT
	//type of this value
	TypeOfValue:IBaseLibrary.TypeClass;
	//pointer to value
	PointerToValue:CommonTypesAndFunctions.ALL_TYPES_UNION_POINTER;
	//Pointer to DB Data
	DB_IN_OUT:POINTER TO DB_IN_OUT;

	
END_VAR
	
THIS^.TypeOfValue:=TypeOfValue;

THIS^.PointerToValue := PointerToValue;

THIS^.SET_DB_IN_OUT_PTR(DB_IN_OUT);

getConfigName := MyName.ReduceToLastNLevels(Level:=2);
END_METHOD

METHOD SET_CONFIG_VALUE_LEVELS
VAR_INPUT
	//type of this value
	TypeOfValue:IBaseLibrary.TypeClass;
	//pointer to value
	PointerToValue:CommonTypesAndFunctions.ALL_TYPES_UNION_POINTER;
	//Pointer to DB Data
	DB_IN_OUT:POINTER TO DB_IN_OUT;
	//Levels
	level:USINT;
END_VAR
	
THIS^.TypeOfValue:=TypeOfValue;

THIS^.PointerToValue := PointerToValue;

THIS^.SET_DB_IN_OUT_PTR(DB_IN_OUT);

getConfigName := MyName.ReduceToLastNLevels(Level:=level);
END_METHOD

PROPERTY SetRealFaktor : uint
SET
RealFaktor:= SetRealFaktor;
END_SET
END_PROPERTY

END_FUNCTION_BLOCK

// MariaDb/Function Blocks/LOGGING_TO_DB_AUTO_ID
FUNCTION_BLOCK LOGGING_TO_DB_AUTO_ID EXTENDS SQL_BASE
VAR_INPUT
	
	Trigger:BOOL;
END_VAR
VAR_OUTPUT
END_VAR
VAR
	BUFFER:ARRAY[0..MyConstants.FB_BUFFER_SIZE] OF LOGGING_DATA;
	
	P_TRIGGER:Standard.R_TRIG;
	N_TRIGGER:Standard.F_TRIG;
	TextOn :STRING(200);
	TextOff :STRING(200);
	IdTextOn:UINT;
	IdTextOff:UINT;
	configDone: BOOL;
	//check config from DB every....s
	CHECK_DB_CONFIG:UINT:=300;
	//var for waiting to check
	CHECK_DB_CONFIG_VAR:UINT;
	//stored Data from request
	DATA_REQUEST:DATA_TO_DB;
	init: BOOL;
	ConfigNameOn:STRING;
	ConfigNameOff:STRING;
	getOn: BOOL;
	getOff: BOOL;
	getOnRequested: BOOL;
	getOffRequested: BOOL;
	steps:UINT;

END_VAR

IF NOT init THEN
	init := TRUE;
	getConfigName := MyName.ReduceToLastNLevels(Level:=2);
	ConfigNameOn := getConfigName;
	ConfigNameOff := getConfigName; 
	ConfigNameOn := CONCAT(STR1:= ConfigNameOn, STR2:= '.TRUE');
	ConfigNameOff := CONCAT(STR1:= ConfigNameOff, STR2:= '.FALSE');
	steps := 1;
END_IF

SQL_NO:=SQL_COMMANDS.WRITE_LOGGING_TEXT;//set SQL no for super^()

SUPER^();
//my work isnt vailid without time... or DB Pointer
IF NOT DbPointerIo THEN RETURN; END_IF
IF NOT DB_IN_OUT^.TIME_IO THEN RETURN; END_IF


//Check if a config request is todo
IF DATA_REQUEST.FB_ID <> 0 AND DB_IN_OUT^.IN.FB_ID = 0 THEN
	DB_IN_OUT^.IN := DATA_REQUEST;
	
	DATA_REQUEST.FB_ID := 0;//delete request
END_IF

CHECK_DATA_FROM_DB();
SET_DB_REQUEST_FOR_TEXT_CONFIG();

P_TRIGGER(CLK:= Trigger);
N_TRIGGER(CLK:= Trigger);

IF BUFFER_INDEX < MyConstants.FB_BUFFER_SIZE AND ((P_TRIGGER.Q AND IdTextOn > 0)OR (N_TRIGGER.Q AND IdTextOff > 0)) AND configDone THEN
	PUSH_LOCAL_BUFFER();
END_IF

METHOD DO_SQL_DATA
VAR_INPUT
END_VAR
SQL_VALUES[0] := GET_STRING_DATE(BUFFER[BUFFER_INDEX].TimeToLog);
IF BUFFER[BUFFER_INDEX].POrN THEN //check if event was positiv or negativ
	SQL_VALUES[1] := TextOn;
	SQL_VALUES[2] := UINT_TO_STRING(IdTextOn);
ELSE
	SQL_VALUES[1] := TextOff;	
	SQL_VALUES[2] := UINT_TO_STRING(IdTextOff);
END_IF
END_METHOD

METHOD PUSH_LOCAL_BUFFER
VAR_INPUT
END_VAR
VAR_IN_OUT
END_VAR
IF BUFFER_INDEX < MyConstants.FB_BUFFER_SIZE - 1 THEN
	BUFFER[BUFFER_INDEX].TimeToLog := DB_IN_OUT^.SYSTEM_TIME;
	BUFFER[BUFFER_INDEX].POrN := Trigger;
END_IF

BUFFER_INDEX := BUFFER_INDEX + 1; 

IF BUFFER_INDEX > MaxBuffer THEN
	MaxBuffer := BUFFER_INDEX;
END_IF
END_METHOD

METHOD PRIVATE CHECK_DATA_FROM_DB
VAR_IN_OUT
END_VAR
VAR
	//DataField Index
	i:UINT;
END_VAR
IF DB_IN_OUT^.OUT.FB_ID = DB_IN_OUT^.FB_NO_AUTO THEN
	//got my request back	
	i := GET_INDEX_DATA_FIELDS_SQL_RESPONSE(src:=ADR(DB_IN_OUT^.OUT.DATA_FROM_DB),SQL_COMMANDS.GET_LOGGING_TEXT);
	IF i = 0 THEN 
	
		SQL_ERROR.SQL_ERROR := 'no data to Sensor';
		
		IF steps = 5 THEN
			steps := 1;
			CHECK_DB_CONFIG_VAR := CHECK_DB_CONFIG + DB_IN_OUT^.FB_NO_AUTO;
			TextOff := '';
			IdTextOff := 0;
			//so create new entry...
			SQL_VALUES[0] := ConfigNameOff;
			SQL_VALUES[1] := ConfigNameOff;
			DATA_REQUEST := PUT_SQL_TO_BUFFER(SQL_NO:=SQL_COMMANDS.CREATE_NEW_TEXT_ENTRY);
		END_IF
		
		IF steps = 3 THEN
			steps := 4;
			TextOn := '';
			IdTextOn := 0;
			//so create new entry...
			SQL_VALUES[0] := ConfigNameOn;
			SQL_VALUES[1] := ConfigNameOn;
			DATA_REQUEST := PUT_SQL_TO_BUFFER(SQL_NO:=SQL_COMMANDS.CREATE_NEW_TEXT_ENTRY); 
		END_IF
		//SQL I.O. but no data 
	ELSE
		IF steps = 5 THEN
			steps := 1;
			CHECK_DB_CONFIG_VAR := CHECK_DB_CONFIG + DB_IN_OUT^.FB_NO_AUTO;
			configDone := TRUE;
			TextOff := GET_STRING_FROM_RESPONSE(SRC:=ADR(DB_IN_OUT^.OUT.DATA_FROM_DB), SIZE:=SIZEOF(DB_IN_OUT^.OUT.DATA_FROM_DB),I:=i);
			IF LEN(STR:= TextOff) > 0 THEN
				IdTextOff := LIMIT(1, STRING_TO_WORD(GET_STRING_FROM_RESPONSE(SRC:=ADR(DB_IN_OUT^.OUT.DATA_FROM_DB), SIZE:=SIZEOF(DB_IN_OUT^.OUT.DATA_FROM_DB),I:=i)), 65000);
			ELSE
				IdTextOff := 0;
			END_IF
			
		END_IF
		IF steps = 3 THEN
			steps := 4;
			TextOn := GET_STRING_FROM_RESPONSE(SRC:=ADR(DB_IN_OUT^.OUT.DATA_FROM_DB), SIZE:=SIZEOF(DB_IN_OUT^.OUT.DATA_FROM_DB),I:=i);
			IF LEN(STR:= TextOn) > 0 THEN 
				IdTextOn := LIMIT(1, STRING_TO_WORD(GET_STRING_FROM_RESPONSE(SRC:=ADR(DB_IN_OUT^.OUT.DATA_FROM_DB), SIZE:=SIZEOF(DB_IN_OUT^.OUT.DATA_FROM_DB),I:=i)), 65000);
			ELSE
				IdTextOn := 0;
			END_IF
		END_IF
		
	END_IF
	DB_IN_OUT^.OUT.FB_ID := 0;//delete response
	
END_IF
END_METHOD

METHOD PRIVATE SET_DB_REQUEST_FOR_TEXT_CONFIG
VAR_IN_OUT
	
END_VAR
//check if time is over
IF CHECK_DB_CONFIG_VAR > 0  THEN
	IF DB_IN_OUT^.IMP THEN
		CHECK_DB_CONFIG_VAR := CHECK_DB_CONFIG_VAR - 1;
	END_IF
	RETURN;	
END_IF
IF NOT DB_IN_OUT^.SQL_CONNECTED THEN RETURN; END_IF
//first get on text
IF steps = 1 THEN
	steps := 2;
END_IF

IF steps = 2 AND DATA_REQUEST.FB_ID = 0 THEN
	SQL_VALUES[0] := ConfigNameOn;
	DATA_REQUEST := PUT_SQL_TO_BUFFER(SQL_NO:=SQL_COMMANDS.GET_LOGGING_TEXT);
	steps := 3;
END_IF

IF steps = 4 AND DATA_REQUEST.FB_ID = 0 THEN
	SQL_VALUES[0] := ConfigNameOff;
	DATA_REQUEST := PUT_SQL_TO_BUFFER(SQL_NO:=SQL_COMMANDS.GET_LOGGING_TEXT);
	steps := 5;
END_IF
END_METHOD

END_FUNCTION_BLOCK

// MariaDb/Function Blocks/VALUE_TO_DB_AUTO_ID_ANY
(*HOWTO
this function controls the sending of process data to DB.
if the queue to db is full it stors the value and date local.
if this local buffer is full, the request is dropt.
the id of the call aof this function must be greater then 0 for detection if the queue to db is empty
This FB creats datapoints by its names
*)


FUNCTION_BLOCK VALUE_TO_DB_AUTO_ID_ANY EXTENDS SQL_BASE
VAR_INPUT

END_VAR
VAR_OUTPUT
END_VAR
VAR_IN_OUT
	
END_VAR
VAR
	//pointer to extern value
	PointerToValue:CommonTypesAndFunctions.ALL_TYPES_UNION_POINTER;
	
	//Value itself
	Value:CommonTypesAndFunctions.ALL_TYPES_UNION;
	//Impulse for value
	ImpValue:BOOL;
	//Value Name
	Name:STRING(50);
	//type of this value
	TypeOfValue:IBaseLibrary.TypeClass;
	//Number of Value in DB
	ValueNum:UINT;
	//stored Data from request
	DATA_REQUEST:DATA_TO_DB;
	//buffer for DB Offline
	BUFFER:ARRAY[0..MyConstants.FB_BUFFER_SIZE] OF VALUE_TO_DB_DATA_OFFLINE;
	

	//Delta time
	DELTA_T:UINT := 60;
	//Time var for DELTA_T
	DELTA_T_VAR:UINT;
	//type of var to save
	VAR_TYPE:UINT;
	//delta value
	DeltaVar:UINT:=1;
	//Last value of VAR send to DB
	LAST_VALUE:CommonTypesAndFunctions.ALL_TYPES_UNION;
	//request by time and Value given
	REQUEST_INSERT: BOOL;
	//Faktor for real for fix komma
	RealFaktor:UINT:=1;
	//check config from DB every....s
	CHECK_DB_CONFIG:UINT:=300;
	//var for waiting to check
	CHECK_DB_CONFIG_VAR:UINT;
	
	FL_IMP_TO_DB:R_TRIG;
	// set to true, if config is reaced
	configDone: BOOL;
	

END_VAR

//set right config status to parent
SQLInvalid := NOT configDone OR valueNum = 0;
SQL_NO:=SQL_COMMANDS.SEND_PW_PROZEDUR;//set SQL no for super^()
SUPER^();
//if not config, then leave, do this after super so we calc correct FB numbers
IF NOT DbPointerIo THEN RETURN; END_IF;


//just work when Time is i.o.
IF NOT DB_IN_OUT^.TIME_IO THEN RETURN; END_IF
//get value from pointer
Value := CommonTypesAndFunctions.GetValueFromPointer(PointerToValue:= PointerToValue, TypeOfValue:= TypeOfValue);
//Check if a config request is todo
IF DATA_REQUEST.FB_ID <> 0 AND DB_IN_OUT^.IN.FB_ID = 0 THEN
	DB_IN_OUT^.IN := DATA_REQUEST;
	
	DATA_REQUEST.FB_ID := 0;//delete request
END_IF

CHECK_DATA_FROM_DB();

//no second imp, nothing to do...
IF NOT DB_IN_OUT^.IMP  THEN
	RETURN;
END_IF
SET_DB_REQUEST_FOR_PW_CONFIG();
//check time over or impulse
FL_IMP_TO_DB(CLK:= ImpValue);
IF DELTA_T_VAR >0 THEN
	DELTA_T_VAR := DELTA_T_VAR -1;
	IF NOT FL_IMP_TO_DB.Q THEN
		RETURN;
	END_IF
END_IF
//check delta V
REQUEST_INSERT := CommonTypesAndFunctions.CheckDeltaValue(Value:= Value, DeltaVar:= DeltaVar, Faktor:= RealFaktor, LastValue:= LAST_VALUE, TypeOfValue:= TypeOfValue);
//nothing todo...
IF NOT REQUEST_INSERT THEN RETURN; END_IF
//we have an request, so first set new intervall
DELTA_T_VAR := DELTA_T - 1;

//push every Data to local buffer, may we lose an cycle but we have only on place to db 
//check buffer to DB free
	//push to lokal buffer
	//if buffer is full drop request
IF BUFFER_INDEX < MyConstants.FB_BUFFER_SIZE THEN
	PUSH_LOCAL_BUFFER();
END_IF

REQUEST_INSERT := FALSE;

METHOD PRIVATE PUSH_LOCAL_BUFFER
VAR_INPUT
END_VAR
VAR_IN_OUT
END_VAR
IF BUFFER_INDEX < MyConstants.FB_BUFFER_SIZE - 1 THEN 
	BUFFER[BUFFER_INDEX].value := Value;
	BUFFER[BUFFER_INDEX].value_time := DB_IN_OUT^.SYSTEM_TIME;
	BUFFER_INDEX := BUFFER_INDEX + 1; 
END_IF
IF BUFFER_INDEX > MaxBuffer THEN
	MaxBuffer := BUFFER_INDEX;
END_IF
END_METHOD

METHOD PRIVATE SET_DB_REQUEST_FOR_PW_CONFIG
VAR_IN_OUT
	
END_VAR
//check if time is over
IF CHECK_DB_CONFIG_VAR > 0 THEN
	CHECK_DB_CONFIG_VAR := CHECK_DB_CONFIG_VAR - 1;
	RETURN;	
END_IF
IF NOT DB_IN_OUT^.SQL_CONNECTED THEN RETURN; END_IF
//set new intervall
CHECK_DB_CONFIG_VAR := CHECK_DB_CONFIG + DB_IN_OUT^.FB_NO_AUTO;
//now put the request to DB
SQL_VALUES[0] := getConfigName;
DATA_REQUEST := PUT_SQL_TO_BUFFER(SQL_NO:=SQL_COMMANDS.SEND_REQUEST_GET_PW_CONFIG_INSTANCE_NAME);
END_METHOD

METHOD PRIVATE CHECK_DATA_FROM_DB
VAR_IN_OUT
END_VAR
VAR
	//DataField Index
	i:UINT;
END_VAR
IF DB_IN_OUT^.OUT.FB_ID = DB_IN_OUT^.FB_NO_AUTO THEN
	//got my request back	
	i := GET_INDEX_DATA_FIELDS_SQL_RESPONSE(src:=ADR(DB_IN_OUT^.OUT.DATA_FROM_DB),SQL_COMMANDS.SEND_REQUEST_GET_PW_CONFIG_INSTANCE_NAME);
	IF i = 0 THEN 
	
		SQL_ERROR.SQL_ERROR := 'no data to Sensor';
		//so create new entry...
		SQL_VALUES[0] := getConfigName;
		SQL_VALUES[1] := getConfigName;
		SQL_VALUES[2] := TO_STRING(RealFaktor);
		DATA_REQUEST := PUT_SQL_TO_BUFFER(SQL_NO:=SQL_COMMANDS.CREATE_NEW_SENSOR_ENTRY);
		//SQL I.O. but no data 
	ELSE
		//parse first data
		DELTA_T := LIMIT(1, STRING_TO_WORD(GET_STRING_FROM_RESPONSE(SRC:=ADR(DB_IN_OUT^.OUT.DATA_FROM_DB), SIZE:=SIZEOF(DB_IN_OUT^.OUT.DATA_FROM_DB),I:=i)), 65000);
		//Set var to new value to prevent high times in some cases
		DELTA_T_VAR := LIMIT(1, DELTA_T, DELTA_T_VAR);
		//get faktor for Real values
		RealFaktor := LIMIT(1, STRING_TO_WORD(GET_STRING_FROM_RESPONSE(SRC:=ADR(DB_IN_OUT^.OUT.DATA_FROM_DB), SIZE:=SIZEOF(DB_IN_OUT^.OUT.DATA_FROM_DB),I:=i)),100);
		//get min delta for values
		DeltaVar := LIMIT(1, STRING_TO_WORD(GET_STRING_FROM_RESPONSE(SRC:=ADR(DB_IN_OUT^.OUT.DATA_FROM_DB), SIZE:=SIZEOF(DB_IN_OUT^.OUT.DATA_FROM_DB),I:=i)),1000);
		//Get sensor Num
		ValueNum := LIMIT(1, STRING_TO_WORD(GET_STRING_FROM_RESPONSE(SRC:=ADR(DB_IN_OUT^.OUT.DATA_FROM_DB), SIZE:=SIZEOF(DB_IN_OUT^.OUT.DATA_FROM_DB),I:=i)), 65000);
		configDone := TRUE;
	END_IF
	DB_IN_OUT^.OUT.FB_ID := 0;//delete response
	
END_IF
END_METHOD

METHOD PRIVATE DO_SQL_DATA
VAR_INPUT
END_VAR
SQL_VALUES[0] := GET_STRING_DATE(BUFFER[BUFFER_INDEX].value_time);
SQL_VALUES[1] := UINT_TO_STRING(ValueNum);
SQL_VALUES[2] := CommonTypesAndFunctions.GetValueStringFaktor(VALUE:= BUFFER[BUFFER_INDEX].value, TypeOfValue:= TypeOfValue, RealFaktor:= to_int(RealFaktor), DecimalPlace:= 0);
END_METHOD

METHOD SET_CONFIG_VALUE
VAR_INPUT
	//which var?
	which:ANY;
	//Pointer to DB Data
	DB_IN_OUT:POINTER TO DB_IN_OUT;

	
END_VAR
	
THIS^.TypeOfValue:=TO_INT(which.TypeClass);

THIS^.PointerToValue.POINTER_TO_BYTE_T := which.pValue;

THIS^.SET_DB_IN_OUT_PTR(DB_IN_OUT);

getConfigName := MyName.ReduceToLastNLevels(Level:=2);
END_METHOD

METHOD SET_CONFIG_VALUE_LEVELS
VAR_INPUT
	//which var?
	which:ANY;
	//Pointer to DB Data
	DB_IN_OUT:POINTER TO DB_IN_OUT;
	//Levels
	level:USINT;
END_VAR
THIS^.TypeOfValue:=TO_INT(which.TypeClass);

THIS^.PointerToValue.POINTER_TO_BYTE_T := which.pValue;

THIS^.SET_DB_IN_OUT_PTR(DB_IN_OUT);

getConfigName := MyName.ReduceToLastNLevels(Level:=level);
END_METHOD

END_FUNCTION_BLOCK

// MariaDb/Function Blocks/VALUE_TO_DB_AUTO_ID_JSON
FUNCTION_BLOCK VALUE_TO_DB_AUTO_ID_JSON
VAR_INPUT
END_VAR
VAR_OUTPUT
END_VAR
VAR
	RealFaktor:UINT:=1;
	FbDB:VALUE_TO_DB_AUTO_ID;
	value:CommonTypesAndFunctions.ALL_TYPES_UNION;
	UnionVarType:TypeClass;
	FromVar:POINTER TO PRO_JSON.JSONVAR;
	levels:USINT:=3;
	init: BOOL;

END_VAR

IF NOT init THEN
	init := TRUE;
	FbDB.SetRealFaktor:= RealFaktor;
END_IF
CASE UnionVarType OF
	TYPE_LINT:
		value.LINT_T:= FromVar^.Integer;
	TYPE_LREAL:
		value.LREAL_T:= FromVar^.Number;	
END_CASE
FbDB();

//FB_Init ist immer implizit verfügbar und wird primär für die Initialisierung verwendet.
//Der Rückgabewert wird nicht ausgewertet. Für gezielte Einflussnahme können Sie
//die Methoden explizit deklarieren und darin mit dem Standard-Initialisierungscode 
//zusätzlichen Code bereitstellen. Sie können den Rückgabewert auswerten.
METHOD FB_Init: BOOL
VAR_INPUT    
bInitRetains: BOOL; // TRUE: Die Retain-Variablen werden initialisiert (Reset warm / Reset kalt)    
bInCopyCode: BOOL;  // TRUE: Die Instanz wird danach in den Kopiercode kopiert (Online-Change)
//which var?
which:POINTER TO PRO_JSON.JSONVAR;
//Type of Var
VarType:PRO_JSON.JSONVALUETYPE;
//Pointer to DB Data
DB_IN_OUT:POINTER TO DB_IN_OUT;

	
END_VAR
VAR
	tmpPointer:CommonTypesAndFunctions.ALL_TYPES_UNION_POINTER;
END_VAR
CASE VarType OF
	PRO_JSON.JSONVALUETYPE.json_integer:
		tmpPointer.POINTER_TO_LINT_T := ADR(value.LINT_T);
		UnionVarType:= TYPE_LINT;
	PRO_JSON.JSONVALUETYPE.json_number:
		tmpPointer.POINTER_TO_LREAL_T := ADR(value.LREAL_T);
		UnionVarType:= TYPE_LREAL;
END_CASE
FromVar := which;

FbDB.SET_CONFIG_VALUE_LEVELS(DB_IN_OUT:= DB_IN_OUT, level:= levels, PointerToValue:= tmpPointer, TypeOfValue:= UnionVarType);
END_METHOD

END_FUNCTION_BLOCK

// MariaDb/Function Blocks/COUNTER_DB_AUTO_ID
(*do never ever try to use dynamic divider --> easy count of comsumption is not possible*)
FUNCTION_BLOCK COUNTER_DB_AUTO_ID EXTENDS SQL_BASE
VAR_INPUT
	//impulse from counter
	imp:BOOL;
	//time until usage output goes low due no more imp, but no dadabase action.
	TimeToZero:TIME:=T#5M;
END_VAR
VAR_OUTPUT
	usage:UDINT;
END_VAR
VAR
	//Number of counter in DB
	CounterNum:UINT:=0;
	//rising trigger of counter
	TrRis:Standard.R_TRIG;
	//buffer for DB Offline
	BUFFER:ARRAY[0..MyConstants.FB_BUFFER_SIZE] OF COUNTER_TO_DB_DATA;
	//impulses since start
	imps:ULINT;
	//consumption Factor
	LConsumptionFaktor:UDINT;
	//stored Data from request
	DATA_REQUEST:DATA_TO_DB;
	//var for getting CounterNum
	getCounterNum: BOOL := TRUE;
	//time when we got to zero on usage output
	TimeZero:DT;
END_VAR

//set right config status to parent
SQLInvalid := CounterNum = 0;
SUPER^();
//if not config, then leave, do this after super so we calc correct FB numbers
IF NOT DbPointerIo THEN RETURN; END_IF;

//just work when Time is i.o.
IF NOT DB_IN_OUT^.TIME_IO THEN RETURN; END_IF
//if no counter num and in free, ask for counter num
IF counterNum = 0 AND DB_IN_OUT^.IN.FB_ID = 0 THEN
	SET_DB_REQUEST_FOR_COUNTER_NUM();
END_IF
//always read SQL response due counter usage
CHECK_DATA_FROM_DB();
//Check if a we want to read counter num
IF DATA_REQUEST.FB_ID <> 0 AND DB_IN_OUT^.IN.FB_ID = 0 THEN
	DB_IN_OUT^.IN := DATA_REQUEST;
	
	DATA_REQUEST.FB_ID := 0;//delete request
END_IF
IF TimeZero < DB_IN_OUT^.SYSTEM_TIME THEN
	usage:= 0;
END_IF
TrRis(CLK:= imp);
//do all work only on rising edge
IF NOT TrRis.Q THEN RETURN; END_IF

//update zero time
TimeZero:=  DB_IN_OUT^.SYSTEM_TIME + TimeToZero;

imps := imps + 1;
IF BUFFER_INDEX < MyConstants.FB_BUFFER_SIZE THEN
	PUSH_LOCAL_BUFFER();
END_IF

METHOD SET_CONFIG_COUNTER
VAR_INPUT
	//Pointer to DB Data
	DB_IN_OUT:POINTER TO DB_IN_OUT;
	//factor for DB query
	//if 0 don't calculat actualy usage
	consumptionFaktor:UDINT;
END_VAR
THIS^.SET_DB_IN_OUT_PTR(DB_IN_OUT);

IF consumptionFaktor = 0 THEN
	//set to at least 1
	consumptionFaktor:= 1;
END_IF
LConsumptionFaktor := consumptionFaktor;

	
SQL_NO:=SQL_COMMANDS.SEND_COUNTER_PROZEDUR;//set SQL no for super^()

getConfigName := MyName.ReduceToLastNLevels(Level:=2);
END_METHOD

METHOD PRIVATE PUSH_LOCAL_BUFFER
VAR_INPUT
END_VAR
IF BUFFER_INDEX < MyConstants.FB_BUFFER_SIZE - 1 THEN 
	BUFFER[BUFFER_INDEX].value_time := DB_IN_OUT^.SYSTEM_TIME;
	BUFFER_INDEX := BUFFER_INDEX + 1; 
END_IF
IF BUFFER_INDEX > MaxBuffer THEN
	MaxBuffer := BUFFER_INDEX;
END_IF
END_METHOD

METHOD PRIVATE DO_SQL_DATA
VAR_INPUT
END_VAR
VAR
	i:UINT;
	lowest:UINT;
END_VAR
//BUFFER_INDEX points to last valid value, so search the oldest and get this to DB
IF BUFFER_INDEX = 0 THEN
	//if just one item --> don't care
	SQL_VALUES[0] := GET_STRING_DATE(BUFFER[BUFFER_INDEX].value_time);
ELSE
	lowest:= 0;
	FOR i:= 0 TO BUFFER_INDEX DO
		IF BUFFER[i].value_time < BUFFER[lowest].value_time THEN
			lowest:= i; 
		END_IF
	END_FOR
	SQL_VALUES[0] := GET_STRING_DATE(BUFFER[lowest].value_time);
	//now copy last in lowest for consistens
	BUFFER[lowest].value_time:= BUFFER[BUFFER_INDEX].value_time;
END_IF
SQL_VALUES[1] := UINT_TO_STRING(CounterNum);
SQL_VALUES[2] := UDINT_TO_STRING(LConsumptionFaktor);
END_METHOD

METHOD PRIVATE CHECK_DATA_FROM_DB
VAR_IN_OUT
END_VAR
VAR
	i:UINT;
END_VAR
IF DB_IN_OUT^.OUT.FB_ID = DB_IN_OUT^.FB_NO_AUTO THEN
	//got my request back
	IF DB_IN_OUT^.OUT.SQL_NO = SQL_COMMANDS.GET_COUNTER_NUM THEN
		i := GET_INDEX_DATA_FIELDS_SQL_RESPONSE(src:=ADR(DB_IN_OUT^.OUT.DATA_FROM_DB),SQL_COMMANDS.GET_COUNTER_NUM);
		IF i = 0 THEN 
			//SQL I.O. but no data
			SQL_ERROR.SQL_ERROR := 'no data to Sensor';
			//so create new entry...
			SQL_VALUES[0] := getConfigName;
			SQL_VALUES[1] := getConfigName;
			SQL_VALUES[2] := '1';
			DATA_REQUEST := PUT_SQL_TO_BUFFER(SQL_NO:=SQL_COMMANDS.CREATE_NEW_COUNTER_ENTRY);
			getCounterNum := TRUE;
		ELSE
			//parse first data --> counter num
			CounterNum := LIMIT(1, STRING_TO_WORD(GET_STRING_FROM_RESPONSE(SRC:=ADR(DB_IN_OUT^.OUT.DATA_FROM_DB), SIZE:=SIZEOF(DB_IN_OUT^.OUT.DATA_FROM_DB),I:=i)), 65000);
		END_IF
	END_IF
	IF DB_IN_OUT^.OUT.SQL_NO = SQL_COMMANDS.SEND_COUNTER_PROZEDUR THEN
		i := GET_INDEX_DATA_FIELDS_SQL_RESPONSE(src:=ADR(DB_IN_OUT^.OUT.DATA_FROM_DB),SQL_COMMANDS.GET_COUNTER_NUM);
		IF i > 0 THEN
			usage := LIMIT(1, STRING_TO_WORD(GET_STRING_FROM_RESPONSE(SRC:=ADR(DB_IN_OUT^.OUT.DATA_FROM_DB), SIZE:=SIZEOF(DB_IN_OUT^.OUT.DATA_FROM_DB),I:=i)), 65000);
		END_IF
	END_IF
	DB_IN_OUT^.OUT.FB_ID := 0;//delete response
END_IF
END_METHOD

METHOD PRIVATE SET_DB_REQUEST_FOR_COUNTER_NUM
VAR_IN_OUT
	
END_VAR

IF NOT DB_IN_OUT^.SQL_CONNECTED THEN RETURN; END_IF
IF getCounterNum = TRUE THEN
	getCounterNum := FALSE;
	//now put the request to DB
	SQL_VALUES[0] := getConfigName;
	DATA_REQUEST := PUT_SQL_TO_BUFFER( SQL_NO:=SQL_COMMANDS.GET_COUNTER_NUM);	
END_IF
END_METHOD

END_FUNCTION_BLOCK
